Yaskawa INFORM job: DEMO_ROOF_SIDE_0625_3PAINT_9.JBI

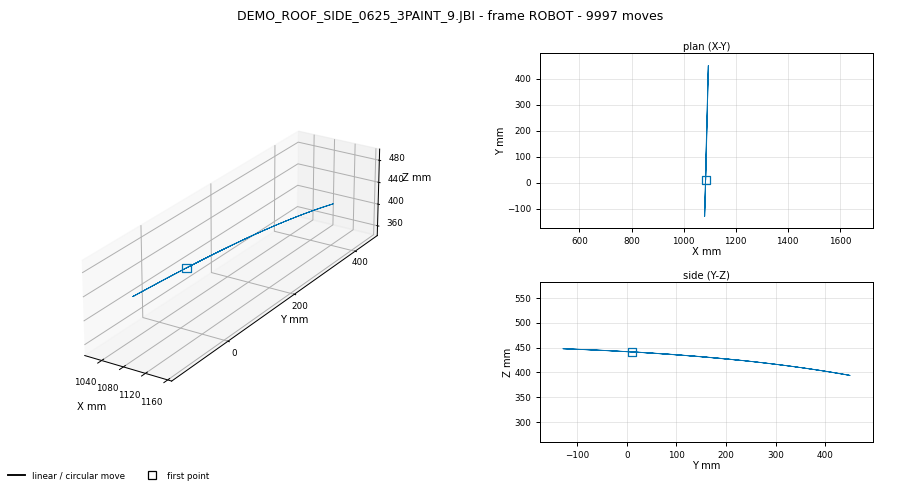
[picture p0: tool path of DEMO_ROOF_SIDE_0625_3PAINT_9.JBI in frame ROBOT, 9997 of 9997 moves have a stored position in this frame; points joined in program order, loops and branches not executed]
/JOB
//NAME DEMO_ROOF_SIDE_0625_3PAINT9
//POS
///NPOS 9997,0,0,0,0,0
///TOOL 0
///USER 0
///POSTYPE ROBOT
///RECTAN
///RCONF 1,0,0,0,0,0,0,0,0,0,0,0,0,0,0,0,0,0,0,0,0,0,0,0
C00000=1085.250,11.093,441.789,174.492,19.107,153.129
C00001=1085.256,11.342,441.774,174.493,19.109,153.129
C00002=1085.262,11.592,441.760,174.496,19.111,153.129
C00003=1085.269,11.841,441.746,174.497,19.113,153.129
C00004=1085.275,12.091,441.732,174.498,19.115,153.129
C00005=1085.280,12.340,441.717,174.500,19.118,153.129
C00006=1085.286,12.590,441.703,174.502,19.119,153.129
C00007=1085.292,12.839,441.688,174.503,19.121,153.129
C00008=1085.298,13.089,441.675,174.505,19.123,153.129
C00009=1085.304,13.338,441.660,174.507,19.125,153.130
C00010=1085.310,13.588,441.646,174.508,19.127,153.130
C00011=1085.315,13.837,441.631,174.509,19.129,153.130
C00012=1085.321,14.087,441.617,174.512,19.131,153.130
C00013=1085.327,14.336,441.602,174.513,19.133,153.130
C00014=1085.333,14.586,441.588,174.514,19.134,153.130
C00015=1085.340,14.863,441.572,174.516,19.137,153.130
C00016=1085.346,15.140,441.555,174.517,19.139,153.130
C00017=1085.352,15.417,441.539,174.520,19.141,153.130
C00018=1085.358,15.693,441.524,174.521,19.143,153.131
C00019=1085.365,15.943,441.509,174.523,19.145,153.131
C00020=1085.370,16.192,441.495,174.524,19.147,153.131
C00021=1085.376,16.443,441.480,174.526,19.149,153.131
C00022=1085.382,16.692,441.465,174.528,19.151,153.131
C00023=1085.387,16.941,441.451,174.529,19.153,153.131
C00024=1085.393,17.191,441.436,174.530,19.155,153.131
C00025=1085.399,17.440,441.422,174.533,19.157,153.131
C00026=1085.405,17.689,441.408,174.534,19.159,153.131
C00027=1085.411,17.939,441.393,174.535,19.161,153.132
C00028=1085.416,18.188,441.378,174.537,19.163,153.132
C00029=1085.422,18.438,441.364,174.539,19.165,153.132
C00030=1085.428,18.687,441.349,174.540,19.167,153.132
C00031=1085.434,18.937,441.334,174.541,19.168,153.132
C00032=1085.440,19.187,441.320,174.544,19.171,153.132
C00033=1085.445,19.436,441.305,174.545,19.173,153.132
C00034=1085.451,19.686,441.290,174.546,19.174,153.132
C00035=1085.457,19.935,441.276,174.548,19.177,153.132
C00036=1085.463,20.185,441.261,174.550,19.178,153.132
C00037=1085.469,20.434,441.247,174.551,19.181,153.133
C00038=1085.474,20.684,441.231,174.553,19.183,153.133
C00039=1085.480,20.933,441.217,174.554,19.185,153.133
C00040=1085.486,21.182,441.203,174.556,19.186,153.133
C00041=1085.491,21.432,441.187,174.558,19.189,153.133
C00042=1085.497,21.681,441.173,174.559,19.191,153.133
C00043=1085.503,21.931,441.158,174.561,19.192,153.133
C00044=1085.509,22.180,441.144,174.563,19.195,153.133
C00045=1085.515,22.430,441.128,174.564,19.196,153.133
C00046=1085.520,22.679,441.114,174.565,19.198,153.134
C00047=1085.527,22.930,441.099,174.568,19.200,153.134
C00048=1085.532,23.179,441.084,174.569,19.202,153.134
C00049=1085.538,23.429,441.069,174.570,19.204,153.134
C00050=1085.544,23.677,441.055,174.572,19.206,153.134
C00051=1085.549,23.927,441.040,174.574,19.208,153.134
C00052=1085.555,24.176,441.025,174.575,19.210,153.134
C00053=1085.561,24.426,441.011,174.577,19.212,153.134
C00054=1085.566,24.676,440.995,174.578,19.214,153.134
C00055=1085.572,24.925,440.981,174.580,19.216,153.135
C00056=1085.578,25.175,440.966,174.582,19.218,153.135
C00057=1085.584,25.424,440.951,174.583,19.220,153.135
C00058=1085.590,25.674,440.936,174.585,19.222,153.135
C00059=1085.596,25.922,440.921,174.587,19.224,153.135
C00060=1085.601,26.172,440.905,174.588,19.226,153.135
C00061=1085.607,26.421,440.891,174.589,19.228,153.135
C00062=1085.613,26.672,440.877,174.592,19.230,153.135
C00063=1085.619,26.922,440.861,174.593,19.232,153.135
C00064=1085.625,27.171,440.847,174.594,19.233,153.135
C00065=1085.630,27.421,440.831,174.596,19.236,153.136
C00066=1085.636,27.670,440.816,174.598,19.237,153.136
C00067=1085.642,27.919,440.801,174.599,19.239,153.136
C00068=1085.647,28.168,440.786,174.601,19.241,153.136
C00069=1085.654,28.418,440.771,174.602,19.243,153.136
C00070=1085.659,28.667,440.756,174.604,19.245,153.136
C00071=1085.665,28.917,440.741,174.606,19.247,153.136
C00072=1085.670,29.166,440.726,174.607,19.249,153.136
C00073=1085.677,29.416,440.711,174.609,19.251,153.136
C00074=1085.682,29.665,440.696,174.611,19.253,153.137
C00075=1085.688,29.915,440.681,174.612,19.255,153.137
C00076=1085.693,30.164,440.666,174.613,19.257,153.137
C00077=1085.700,30.414,440.651,174.616,19.259,153.137
C00078=1085.705,30.664,440.635,174.617,19.261,153.137
C00079=1085.712,30.942,440.618,174.619,19.263,153.137
C00080=1085.718,31.220,440.602,174.620,19.265,153.137
C00081=1085.725,31.498,440.585,174.622,19.268,153.137
C00082=1085.731,31.776,440.568,174.624,19.270,153.137
C00083=1085.736,32.025,440.553,174.626,19.272,153.137
C00084=1085.743,32.275,440.538,174.627,19.274,153.138
C00085=1085.748,32.525,440.522,174.629,19.276,153.138
C00086=1085.754,32.774,440.507,174.631,19.278,153.138
C00087=1085.760,33.023,440.492,174.632,19.279,153.138
C00088=1085.765,33.273,440.476,174.634,19.282,153.138
C00089=1085.771,33.522,440.462,174.636,19.283,153.138
C00090=1085.776,33.772,440.446,174.637,19.285,153.138
C00091=1085.783,34.021,440.431,174.639,19.287,153.138
C00092=1085.788,34.271,440.416,174.640,19.289,153.138
C00093=1085.794,34.520,440.400,174.643,19.291,153.138
C00094=1085.800,34.770,440.385,174.644,19.293,153.139
C00095=1085.806,35.020,440.370,174.645,19.295,153.139
C00096=1085.812,35.268,440.355,174.647,19.298,153.139
C00097=1085.817,35.518,440.339,174.649,19.299,153.139
C00098=1085.822,35.768,440.324,174.650,19.301,153.139
C00099=1085.829,36.017,440.309,174.652,19.303,153.139
C00100=1085.835,36.267,440.293,174.654,19.305,153.139
C00101=1085.840,36.516,440.278,174.655,19.307,153.139
C00102=1085.846,36.766,440.263,174.657,19.309,153.139
C00103=1085.852,37.015,440.247,174.659,19.311,153.139
C00104=1085.858,37.264,440.232,174.661,19.313,153.139
C00105=1085.863,37.514,440.217,174.662,19.315,153.140
C00106=1085.870,37.764,440.202,174.663,19.316,153.140
C00107=1085.875,38.012,440.186,174.666,19.319,153.140
C00108=1085.881,38.262,440.170,174.667,19.320,153.140
C00109=1085.886,38.512,440.155,174.668,19.322,153.140
C00110=1085.893,38.760,440.139,174.671,19.324,153.140
C00111=1085.898,39.010,440.124,174.672,19.326,153.140
C00112=1085.904,39.260,440.108,174.674,19.328,153.140
C00113=1085.909,39.509,440.092,174.675,19.330,153.140
C00114=1085.915,39.759,440.077,174.677,19.332,153.140
C00115=1085.921,40.009,440.062,174.679,19.334,153.141
C00116=1085.927,40.257,440.046,174.680,19.336,153.141
C00117=1085.932,40.507,440.030,174.682,19.338,153.141
C00118=1085.938,40.757,440.015,174.684,19.340,153.141
C00119=1085.944,41.006,440.000,174.685,19.342,153.141
C00120=1085.950,41.256,439.984,174.687,19.344,153.141
C00121=1085.955,41.506,439.968,174.688,19.346,153.141
C00122=1085.961,41.754,439.953,174.690,19.348,153.141
C00123=1085.966,42.004,439.937,174.692,19.350,153.141
C00124=1085.972,42.253,439.921,174.693,19.352,153.141
C00125=1085.978,42.502,439.906,174.695,19.354,153.142
C00126=1085.984,42.752,439.890,174.697,19.356,153.142
C00127=1085.990,43.002,439.874,174.698,19.357,153.142
C00128=1085.995,43.252,439.859,174.700,19.360,153.142
C00129=1086.001,43.500,439.843,174.702,19.361,153.142
C00130=1086.007,43.750,439.828,174.704,19.364,153.142
C00131=1086.013,43.999,439.812,174.705,19.365,153.142
C00132=1086.018,44.249,439.797,174.707,19.367,153.142
C00133=1086.024,44.498,439.780,174.709,19.369,153.142
C00134=1086.030,44.748,439.765,174.710,19.371,153.142
C00135=1086.035,44.997,439.749,174.712,19.373,153.142
C00136=1086.041,45.247,439.733,174.714,19.375,153.143
C00137=1086.047,45.496,439.717,174.715,19.377,153.143
C00138=1086.052,45.746,439.702,174.717,19.379,153.143
C00139=1086.058,45.995,439.686,174.719,19.381,153.143
C00140=1086.063,46.245,439.670,174.721,19.383,153.143
C00141=1086.069,46.494,439.654,174.722,19.385,153.143
C00142=1086.074,46.743,439.639,174.723,19.387,153.143
C00143=1086.081,47.022,439.621,174.726,19.389,153.143
C00144=1086.087,47.300,439.603,174.728,19.391,153.143
C00145=1086.092,47.578,439.585,174.729,19.393,153.144
C00146=1086.100,47.857,439.568,174.731,19.396,153.144
C00147=1086.105,48.105,439.552,174.733,19.398,153.144
C00148=1086.111,48.355,439.535,174.735,19.400,153.144
C00149=1086.117,48.605,439.520,174.736,19.402,153.144
C00150=1086.123,48.854,439.504,174.738,19.404,153.144
C00151=1086.127,49.103,439.487,174.740,19.406,153.144
C00152=1086.133,49.353,439.472,174.742,19.408,153.144
C00153=1086.139,49.602,439.455,174.743,19.410,153.144
C00154=1086.144,49.852,439.440,174.745,19.411,153.144
C00155=1086.150,50.102,439.424,174.747,19.413,153.144
C00156=1086.156,50.350,439.408,174.748,19.415,153.145
C00157=1086.161,50.600,439.392,174.750,19.417,153.145
C00158=1086.167,50.850,439.376,174.752,19.419,153.145
C00159=1086.173,51.099,439.360,174.753,19.421,153.145
C00160=1086.179,51.348,439.343,174.755,19.423,153.145
C00161=1086.184,51.598,439.328,174.757,19.425,153.145
C00162=1086.190,51.847,439.312,174.759,19.427,153.145
C00163=1086.196,52.096,439.296,174.760,19.429,153.145
C00164=1086.202,52.346,439.279,174.762,19.431,153.145
C00165=1086.207,52.596,439.263,174.764,19.433,153.145
C00166=1086.212,52.845,439.247,174.765,19.434,153.145
C00167=1086.218,53.094,439.231,174.767,19.436,153.145
C00168=1086.224,53.343,439.215,174.769,19.438,153.146
C00169=1086.230,53.593,439.199,174.771,19.440,153.146
C00170=1086.236,53.843,439.183,174.772,19.442,153.146
C00171=1086.242,54.092,439.167,174.774,19.444,153.146
C00172=1086.248,54.341,439.151,174.776,19.446,153.146
C00173=1086.253,54.590,439.135,174.777,19.447,153.146
C00174=1086.258,54.840,439.119,174.779,19.450,153.146
C00175=1086.264,55.089,439.102,174.781,19.451,153.146
C00176=1086.270,55.339,439.086,174.783,19.454,153.146
C00177=1086.276,55.588,439.070,174.784,19.455,153.146
C00178=1086.282,55.838,439.054,174.787,19.457,153.146
C00179=1086.288,56.087,439.037,174.788,19.460,153.146
C00180=1086.293,56.337,439.022,174.789,19.461,153.146
C00181=1086.299,56.587,439.005,174.792,19.463,153.146
C00182=1086.305,56.836,438.989,174.793,19.465,153.146
C00183=1086.310,57.085,438.973,174.795,19.467,153.147
C00184=1086.316,57.334,438.956,174.797,19.469,153.147
C00185=1086.322,57.583,438.940,174.799,19.471,153.147
C00186=1086.328,57.833,438.924,174.800,19.473,153.147
C00187=1086.333,58.082,438.907,174.802,19.474,153.147
C00188=1086.339,58.332,438.891,174.804,19.476,153.147
C00189=1086.345,58.581,438.875,174.805,19.478,153.147
C00190=1086.351,58.830,438.858,174.808,19.480,153.147
C00191=1086.357,59.080,438.842,174.809,19.482,153.147
C00192=1086.362,59.329,438.825,174.811,19.484,153.147
C00193=1086.368,59.579,438.809,174.813,19.486,153.147
C00194=1086.374,59.828,438.793,174.814,19.487,153.147
C00195=1086.380,60.077,438.776,174.816,19.489,153.147
C00196=1086.386,60.327,438.760,174.818,19.491,153.147
C00197=1086.391,60.576,438.743,174.820,19.493,153.148
C00198=1086.397,60.826,438.727,174.821,19.495,153.148
C00199=1086.403,61.075,438.711,174.824,19.497,153.148
C00200=1086.409,61.324,438.695,174.825,19.498,153.148
C00201=1086.415,61.574,438.678,174.827,19.501,153.148
C00202=1086.420,61.823,438.661,174.829,19.502,153.148
C00203=1086.426,62.073,438.645,174.830,19.504,153.148
C00204=1086.432,62.322,438.629,174.832,19.506,153.148
C00205=1086.438,62.571,438.613,174.834,19.507,153.148
C00206=1086.443,62.821,438.596,174.836,19.510,153.148
C00207=1086.451,63.099,438.578,174.838,19.512,153.148
C00208=1086.457,63.376,438.559,174.840,19.513,153.148
C00209=1086.463,63.655,438.541,174.842,19.516,153.148
C00210=1086.470,63.933,438.523,174.844,19.518,153.148
C00211=1086.476,64.182,438.506,174.845,19.519,153.148
C00212=1086.481,64.432,438.489,174.848,19.521,153.148
C00213=1086.487,64.681,438.473,174.849,19.523,153.149
C00214=1086.492,64.930,438.456,174.851,19.525,153.149
C00215=1086.498,65.180,438.439,174.853,19.527,153.149
C00216=1086.504,65.429,438.423,174.855,19.529,153.149
C00217=1086.509,65.679,438.406,174.856,19.531,153.149
C00218=1086.515,65.928,438.390,174.858,19.532,153.149
C00219=1086.521,66.177,438.372,174.860,19.534,153.149
C00220=1086.527,66.426,438.356,174.862,19.536,153.149
C00221=1086.532,66.676,438.339,174.864,19.538,153.149
C00222=1086.538,66.925,438.323,174.865,19.540,153.149
C00223=1086.544,67.175,438.307,174.867,19.542,153.149
C00224=1086.550,67.424,438.289,174.869,19.543,153.149
C00225=1086.556,67.674,438.273,174.871,19.545,153.149
C00226=1086.561,67.923,438.256,174.872,19.547,153.149
C00227=1086.567,68.173,438.240,174.875,19.549,153.149
C00228=1086.573,68.422,438.222,174.876,19.551,153.149
C00229=1086.579,68.671,438.206,174.878,19.553,153.149
C00230=1086.584,68.921,438.189,174.880,19.554,153.149
C00231=1086.590,69.170,438.172,174.882,19.557,153.150
C00232=1086.595,69.419,438.155,174.883,19.558,153.150
C00233=1086.601,69.669,438.139,174.885,19.560,153.150
C00234=1086.607,69.918,438.121,174.887,19.562,153.150
C00235=1086.612,70.167,438.104,174.889,19.564,153.150
C00236=1086.618,70.417,438.088,174.891,19.566,153.150
C00237=1086.624,70.666,438.071,174.892,19.568,153.150
C00238=1086.629,70.915,438.054,174.895,19.570,153.150
C00239=1086.635,71.165,438.037,174.896,19.571,153.150
C00240=1086.641,71.414,438.020,174.898,19.573,153.150
C00241=1086.647,71.664,438.003,174.900,19.575,153.150
C00242=1086.652,71.913,437.986,174.902,19.577,153.150
C00243=1086.658,72.162,437.969,174.903,19.579,153.150
C00244=1086.663,72.412,437.953,174.906,19.581,153.150
C00245=1086.669,72.661,437.935,174.907,19.582,153.150
C00246=1086.675,72.910,437.919,174.909,19.585,153.150
C00247=1086.680,73.159,437.901,174.911,19.586,153.150
C00248=1086.686,73.409,437.884,174.913,19.588,153.150
C00249=1086.692,73.658,437.867,174.914,19.590,153.151
C00250=1086.698,73.908,437.850,174.917,19.592,153.151
C00251=1086.703,74.158,437.833,174.918,19.593,153.151
C00252=1086.709,74.406,437.816,174.921,19.595,153.151
C00253=1086.714,74.656,437.799,174.922,19.597,153.151
C00254=1086.720,74.905,437.782,174.924,19.599,153.151
C00255=1086.726,75.154,437.766,174.926,19.601,153.151
C00256=1086.732,75.404,437.748,174.928,19.603,153.151
C00257=1086.737,75.654,437.731,174.929,19.604,153.151
C00258=1086.743,75.902,437.714,174.932,19.606,153.151
C00259=1086.749,76.152,437.696,174.933,19.608,153.151
C00260=1086.754,76.401,437.679,174.935,19.610,153.151
C00261=1086.760,76.650,437.663,174.937,19.612,153.151
C00262=1086.766,76.900,437.645,174.939,19.614,153.151
C00263=1086.772,77.149,437.628,174.940,19.615,153.151
C00264=1086.777,77.399,437.611,174.943,19.617,153.151
C00265=1086.783,77.648,437.594,174.944,19.619,153.151
C00266=1086.789,77.897,437.576,174.947,19.621,153.151
C00267=1086.795,78.147,437.559,174.948,19.622,153.151
C00268=1086.800,78.396,437.542,174.950,19.624,153.151
C00269=1086.806,78.646,437.525,174.952,19.626,153.151
C00270=1086.812,78.895,437.508,174.954,19.628,153.151
C00271=1086.818,79.173,437.488,174.956,19.630,153.151
C00272=1086.824,79.450,437.469,174.958,19.632,153.152
C00273=1086.830,79.728,437.450,174.960,19.634,153.152
C00274=1086.836,80.007,437.430,174.962,19.636,153.152
C00275=1086.843,80.256,437.413,174.964,19.637,153.152
C00276=1086.848,80.505,437.396,174.966,19.640,153.152
C00277=1086.853,80.754,437.379,174.967,19.641,153.152
C00278=1086.859,81.003,437.361,174.970,19.643,153.152
C00279=1086.865,81.253,437.343,174.972,19.645,153.152
C00280=1086.870,81.503,437.327,174.973,19.647,153.152
C00281=1086.876,81.752,437.309,174.976,19.649,153.152
C00282=1086.881,82.001,437.291,174.977,19.650,153.152
C00283=1086.887,82.251,437.273,174.979,19.652,153.152
C00284=1086.893,82.500,437.257,174.981,19.654,153.152
C00285=1086.898,82.749,437.239,174.983,19.656,153.152
C00286=1086.904,82.998,437.222,174.985,19.657,153.152
C00287=1086.910,83.247,437.205,174.987,19.659,153.152
C00288=1086.916,83.497,437.187,174.988,19.661,153.152
C00289=1086.921,83.747,437.170,174.991,19.663,153.152
C00290=1086.927,83.996,437.152,174.992,19.665,153.152
C00291=1086.933,84.245,437.134,174.994,19.667,153.152
C00292=1086.938,84.494,437.117,174.996,19.668,153.152
C00293=1086.944,84.743,437.099,174.998,19.670,153.152
C00294=1086.949,84.992,437.082,175.000,19.672,153.152
C00295=1086.955,85.243,437.064,175.002,19.674,153.152
C00296=1086.961,85.492,437.047,175.003,19.675,153.152
C00297=1086.966,85.741,437.029,175.006,19.677,153.152
C00298=1086.972,85.990,437.012,175.007,19.679,153.152
C00299=1086.978,86.240,436.994,175.009,19.681,153.152
C00300=1086.983,86.489,436.976,175.012,19.683,153.152
C00301=1086.989,86.738,436.959,175.013,19.684,153.153
C00302=1086.995,86.987,436.941,175.016,19.686,153.152
C00303=1087.000,87.237,436.924,175.017,19.687,153.152
C00304=1087.006,87.486,436.906,175.020,19.689,153.152
C00305=1087.012,87.736,436.888,175.021,19.691,153.153
C00306=1087.017,87.985,436.871,175.023,19.693,153.153
C00307=1087.023,88.234,436.853,175.025,19.694,153.153
C00308=1087.029,88.484,436.835,175.027,19.696,153.153
C00309=1087.035,88.733,436.818,175.029,19.698,153.153
C00310=1087.040,88.982,436.800,175.031,19.700,153.153
C00311=1087.046,89.232,436.782,175.032,19.701,153.153
C00312=1087.052,89.481,436.765,175.035,19.703,153.153
C00313=1087.058,89.730,436.747,175.037,19.705,153.153
C00314=1087.063,89.979,436.729,175.039,19.707,153.153
C00315=1087.069,90.228,436.712,175.041,19.708,153.153
C00316=1087.075,90.478,436.694,175.043,19.710,153.153
C00317=1087.080,90.727,436.676,175.045,19.712,153.153
C00318=1087.087,90.977,436.658,175.046,19.713,153.153
C00319=1087.092,91.226,436.641,175.049,19.715,153.153
C00320=1087.097,91.475,436.622,175.050,19.717,153.153
C00321=1087.103,91.724,436.604,175.052,19.719,153.153
C00322=1087.109,91.973,436.586,175.055,19.721,153.153
C00323=1087.114,92.223,436.569,175.056,19.722,153.153
C00324=1087.120,92.472,436.551,175.059,19.724,153.153
C00325=1087.125,92.722,436.532,175.060,19.726,153.153
C00326=1087.131,92.971,436.515,175.062,19.728,153.153
C00327=1087.137,93.220,436.497,175.064,19.729,153.153
C00328=1087.142,93.469,436.479,175.066,19.731,153.153
C00329=1087.148,93.718,436.461,175.068,19.732,153.153
C00330=1087.154,93.968,436.443,175.070,19.734,153.153
C00331=1087.159,94.217,436.425,175.072,19.736,153.153
C00332=1087.165,94.467,436.407,175.074,19.738,153.153
C00333=1087.170,94.716,436.389,175.076,19.740,153.153
C00334=1087.176,94.965,436.371,175.078,19.741,153.153
C00335=1087.182,95.243,436.351,175.080,19.743,153.153
C00336=1087.188,95.521,436.331,175.082,19.745,153.153
C00337=1087.195,95.799,436.311,175.085,19.747,153.153
C00338=1087.202,96.077,436.290,175.087,19.749,153.153
C00339=1087.206,96.327,436.272,175.088,19.751,153.153
C00340=1087.212,96.576,436.255,175.091,19.752,153.153
C00341=1087.218,96.825,436.236,175.092,19.754,153.153
C00342=1087.224,97.074,436.219,175.095,19.756,153.153
C00343=1087.229,97.324,436.200,175.097,19.758,153.153
C00344=1087.235,97.572,436.182,175.099,19.759,153.153
C00345=1087.241,97.822,436.164,175.101,19.761,153.153
C00346=1087.246,98.071,436.146,175.103,19.762,153.153
C00347=1087.252,98.321,436.127,175.105,19.764,153.153
C00348=1087.258,98.570,436.109,175.107,19.766,153.153
C00349=1087.263,98.820,436.091,175.109,19.768,153.153
C00350=1087.269,99.068,436.073,175.111,19.769,153.153
C00351=1087.275,99.318,436.055,175.113,19.771,153.153
C00352=1087.281,99.567,436.037,175.115,19.773,153.153
C00353=1087.287,99.816,436.018,175.117,19.774,153.153
C00354=1087.292,100.065,436.000,175.119,19.776,153.153
C00355=1087.298,100.315,435.982,175.121,19.778,153.153
C00356=1087.303,100.564,435.963,175.123,19.779,153.153
C00357=1087.309,100.814,435.946,175.125,19.781,153.153
C00358=1087.314,101.062,435.927,175.127,19.782,153.153
C00359=1087.321,101.312,435.909,175.129,19.784,153.153
C00360=1087.326,101.561,435.891,175.132,19.786,153.153
C00361=1087.332,101.811,435.872,175.133,19.788,153.153
C00362=1087.337,102.060,435.854,175.135,19.790,153.153
C00363=1087.343,102.309,435.835,175.137,19.791,153.153
C00364=1087.349,102.558,435.818,175.139,19.793,153.153
C00365=1087.354,102.807,435.798,175.142,19.795,153.153
C00366=1087.360,103.057,435.781,175.143,19.796,153.153
C00367=1087.365,103.306,435.761,175.145,19.798,153.153
C00368=1087.371,103.555,435.744,175.147,19.799,153.153
C00369=1087.377,103.804,435.725,175.150,19.801,153.153
C00370=1087.381,104.054,435.707,175.152,19.803,153.153
C00371=1087.388,104.303,435.688,175.153,19.804,153.153
C00372=1087.393,104.552,435.670,175.156,19.806,153.153
C00373=1087.399,104.801,435.651,175.157,19.807,153.153
C00374=1087.404,105.051,435.633,175.160,19.809,153.153
C00375=1087.410,105.300,435.614,175.162,19.811,153.153
C00376=1087.416,105.549,435.595,175.164,19.812,153.153
C00377=1087.421,105.798,435.577,175.166,19.814,153.153
C00378=1087.427,106.048,435.558,175.167,19.816,153.153
C00379=1087.432,106.297,435.540,175.170,19.817,153.153
C00380=1087.438,106.546,435.521,175.172,19.819,153.153
C00381=1087.444,106.796,435.502,175.174,19.821,153.153
C00382=1087.450,107.045,435.485,175.176,19.822,153.153
C00383=1087.455,107.294,435.465,175.178,19.824,153.153
C00384=1087.461,107.543,435.448,175.180,19.826,153.153
C00385=1087.466,107.793,435.429,175.183,19.827,153.153
C00386=1087.472,108.042,435.409,175.184,19.829,153.153
C00387=1087.478,108.291,435.392,175.187,19.831,153.153
C00388=1087.483,108.540,435.372,175.189,19.832,153.152
C00389=1087.489,108.789,435.354,175.191,19.834,153.153
C00390=1087.495,109.038,435.335,175.193,19.836,153.153
C00391=1087.500,109.288,435.316,175.195,19.837,153.152
C00392=1087.506,109.537,435.298,175.197,19.839,153.152
C00393=1087.512,109.786,435.279,175.199,19.840,153.152
C00394=1087.518,110.036,435.261,175.201,19.842,153.152
C00395=1087.523,110.285,435.242,175.203,19.844,153.152
C00396=1087.529,110.534,435.223,175.206,19.845,153.152
C00397=1087.535,110.783,435.204,175.207,19.847,153.152
C00398=1087.540,111.033,435.186,175.210,19.848,153.152
C00399=1087.546,111.311,435.164,175.212,19.850,153.152
C00400=1087.553,111.589,435.144,175.215,19.852,153.152
C00401=1087.559,111.866,435.123,175.217,19.854,153.152
C00402=1087.566,112.145,435.102,175.219,19.856,153.152
C00403=1087.571,112.394,435.083,175.221,19.857,153.152
C00404=1087.577,112.643,435.064,175.223,19.859,153.152
C00405=1087.582,112.893,435.045,175.225,19.860,153.152
C00406=1087.588,113.141,435.026,175.227,19.862,153.152
C00407=1087.594,113.390,435.007,175.230,19.864,153.152
C00408=1087.599,113.640,434.989,175.231,19.865,153.152
C00409=1087.605,113.890,434.969,175.234,19.867,153.152
C00410=1087.611,114.138,434.951,175.236,19.869,153.152
C00411=1087.616,114.388,434.932,175.238,19.870,153.152
C00412=1087.622,114.637,434.913,175.240,19.872,153.152
C00413=1087.627,114.886,434.894,175.243,19.873,153.152
C00414=1087.633,115.135,434.875,175.244,19.875,153.152
C00415=1087.638,115.385,434.855,175.247,19.877,153.152
C00416=1087.644,115.634,434.836,175.249,19.878,153.152
C00417=1087.649,115.883,434.817,175.251,19.880,153.152
C00418=1087.655,116.132,434.798,175.253,19.882,153.152
C00419=1087.660,116.381,434.779,175.255,19.883,153.152
C00420=1087.666,116.631,434.760,175.257,19.885,153.152
C00421=1087.671,116.880,434.741,175.259,19.886,153.151
C00422=1087.676,117.129,434.722,175.262,19.888,153.151
C00423=1087.682,117.378,434.702,175.263,19.890,153.152
C00424=1087.689,117.627,434.684,175.266,19.891,153.151
C00425=1087.694,117.876,434.665,175.268,19.893,153.151
C00426=1087.699,118.125,434.646,175.270,19.894,153.151
C00427=1087.705,118.375,434.626,175.272,19.896,153.151
C00428=1087.711,118.624,434.607,175.275,19.897,153.151
C00429=1087.716,118.873,434.588,175.276,19.899,153.151
C00430=1087.721,119.122,434.569,175.279,19.900,153.151
C00431=1087.727,119.372,434.550,175.281,19.902,153.151
C00432=1087.733,119.621,434.531,175.283,19.903,153.151
C00433=1087.738,119.870,434.512,175.285,19.905,153.151
C00434=1087.744,120.120,434.492,175.288,19.907,153.151
C00435=1087.749,120.369,434.473,175.289,19.908,153.151
C00436=1087.755,120.618,434.454,175.292,19.910,153.151
C00437=1087.760,120.866,434.434,175.294,19.912,153.151
C00438=1087.766,121.116,434.415,175.296,19.913,153.151
C00439=1087.772,121.365,434.396,175.298,19.915,153.151
C00440=1087.777,121.615,434.377,175.301,19.916,153.151
C00441=1087.782,121.864,434.357,175.302,19.918,153.151
C00442=1087.788,122.113,434.338,175.305,19.919,153.151
C00443=1087.793,122.362,434.318,175.307,19.921,153.151
C00444=1087.799,122.612,434.299,175.309,19.922,153.151
C00445=1087.805,122.861,434.280,175.311,19.924,153.151
C00446=1087.811,123.110,434.260,175.314,19.926,153.150
C00447=1087.816,123.358,434.241,175.315,19.927,153.150
C00448=1087.822,123.608,434.221,175.318,19.929,153.150
C00449=1087.827,123.857,434.202,175.320,19.930,153.150
C00450=1087.833,124.107,434.183,175.322,19.932,153.150
C00451=1087.839,124.356,434.163,175.324,19.933,153.150
C00452=1087.845,124.605,434.144,175.327,19.935,153.150
C00453=1087.850,124.854,434.125,175.329,19.937,153.150
C00454=1087.855,125.103,434.106,175.331,19.938,153.150
C00455=1087.861,125.352,434.086,175.333,19.940,153.150
C00456=1087.867,125.601,434.066,175.336,19.941,153.150
C00457=1087.872,125.851,434.047,175.337,19.942,153.150
C00458=1087.878,126.100,434.027,175.340,19.944,153.150
C00459=1087.884,126.349,434.007,175.342,19.946,153.150
C00460=1087.889,126.599,433.988,175.344,19.947,153.150
C00461=1087.895,126.848,433.968,175.346,19.949,153.150
C00462=1087.901,127.096,433.949,175.349,19.950,153.149
C00463=1087.907,127.375,433.927,175.351,19.952,153.149
C00464=1087.914,127.653,433.906,175.354,19.954,153.149
C00465=1087.920,127.930,433.884,175.356,19.955,153.149
C00466=1087.926,128.208,433.862,175.359,19.957,153.149
C00467=1087.931,128.458,433.842,175.361,19.959,153.149
C00468=1087.937,128.707,433.822,175.363,19.960,153.149
C00469=1087.943,128.956,433.803,175.365,19.961,153.149
C00470=1087.949,129.206,433.783,175.368,19.963,153.149
C00471=1087.955,129.454,433.763,175.369,19.964,153.149
C00472=1087.960,129.704,433.744,175.372,19.965,153.149
C00473=1087.966,129.953,433.724,175.375,19.967,153.149
C00474=1087.971,130.202,433.704,175.377,19.968,153.148
C00475=1087.977,130.451,433.684,175.379,19.970,153.148
C00476=1087.983,130.701,433.665,175.381,19.971,153.148
C00477=1087.989,130.950,433.645,175.384,19.973,153.148
C00478=1087.995,131.199,433.626,175.385,19.974,153.148
C00479=1088.000,131.448,433.605,175.388,19.975,153.148
C00480=1088.006,131.697,433.585,175.390,19.977,153.148
C00481=1088.012,131.946,433.566,175.393,19.979,153.148
C00482=1088.018,132.195,433.546,175.395,19.980,153.148
C00483=1088.023,132.445,433.527,175.397,19.981,153.148
C00484=1088.029,132.694,433.506,175.400,19.983,153.148
C00485=1088.034,132.943,433.487,175.401,19.984,153.148
C00486=1088.040,133.192,433.467,175.404,19.986,153.147
C00487=1088.046,133.441,433.447,175.406,19.987,153.147
C00488=1088.051,133.690,433.427,175.409,19.989,153.147
C00489=1088.057,133.940,433.407,175.410,19.990,153.147
C00490=1088.063,134.188,433.387,175.413,19.992,153.147
C00491=1088.067,134.438,433.367,175.416,19.993,153.147
C00492=1088.073,134.687,433.347,175.418,19.995,153.147
C00493=1088.079,134.936,433.327,175.420,19.996,153.147
C00494=1088.084,135.186,433.307,175.422,19.998,153.147
C00495=1088.090,135.434,433.287,175.425,19.999,153.147
C00496=1088.096,135.683,433.267,175.427,20.001,153.147
C00497=1088.101,135.933,433.248,175.429,20.002,153.147
C00498=1088.107,136.182,433.228,175.431,20.004,153.146
C00499=1088.113,136.431,433.207,175.434,20.005,153.146
C00500=1088.119,136.680,433.187,175.436,20.007,153.146
C00501=1088.124,136.929,433.167,175.438,20.008,153.146
C00502=1088.130,137.178,433.147,175.440,20.010,153.146
C00503=1088.135,137.427,433.127,175.443,20.011,153.146
C00504=1088.141,137.676,433.107,175.446,20.013,153.146
C00505=1088.146,137.926,433.088,175.447,20.014,153.146
C00506=1088.152,138.175,433.067,175.450,20.015,153.146
C00507=1088.158,138.424,433.047,175.452,20.017,153.146
C00508=1088.163,138.673,433.027,175.455,20.019,153.146
C00509=1088.169,138.921,433.007,175.456,20.020,153.146
C00510=1088.174,139.171,432.986,175.459,20.021,153.145
C00511=1088.180,139.420,432.967,175.462,20.022,153.145
C00512=1088.185,139.669,432.946,175.464,20.024,153.145
C00513=1088.190,139.918,432.926,175.466,20.025,153.145
C00514=1088.197,140.168,432.905,175.468,20.026,153.145
C00515=1088.202,140.417,432.885,175.471,20.028,153.145
C00516=1088.208,140.666,432.865,175.473,20.030,153.145
C00517=1088.214,140.915,432.844,175.475,20.031,153.145
C00518=1088.220,141.164,432.824,175.478,20.032,153.145
C00519=1088.225,141.413,432.804,175.480,20.034,153.144
C00520=1088.230,141.663,432.784,175.483,20.035,153.144
C00521=1088.236,141.911,432.764,175.485,20.037,153.144
C00522=1088.241,142.160,432.743,175.487,20.038,153.144
C00523=1088.246,142.410,432.723,175.489,20.040,153.144
C00524=1088.253,142.659,432.703,175.492,20.041,153.144
C00525=1088.258,142.908,432.682,175.494,20.043,153.144
C00526=1088.263,143.157,432.661,175.496,20.044,153.144
C00527=1088.270,143.435,432.639,175.499,20.046,153.144
C00528=1088.276,143.713,432.616,175.502,20.047,153.144
C00529=1088.282,143.990,432.593,175.505,20.049,153.143
C00530=1088.289,144.268,432.570,175.507,20.050,153.143
C00531=1088.295,144.518,432.550,175.510,20.052,153.143
C00532=1088.300,144.767,432.529,175.511,20.053,153.143
C00533=1088.306,145.016,432.509,175.514,20.055,153.143
C00534=1088.311,145.265,432.489,175.516,20.056,153.143
C00535=1088.316,145.514,432.468,175.519,20.058,153.143
C00536=1088.322,145.763,432.448,175.521,20.059,153.143
C00537=1088.328,146.013,432.427,175.523,20.060,153.143
C00538=1088.333,146.262,432.407,175.526,20.062,153.143
C00539=1088.339,146.511,432.386,175.528,20.063,153.142
C00540=1088.345,146.759,432.365,175.531,20.065,153.142
C00541=1088.350,147.008,432.345,175.533,20.066,153.142
C00542=1088.356,147.258,432.324,175.535,20.067,153.142
C00543=1088.362,147.507,432.304,175.538,20.069,153.142
C00544=1088.367,147.756,432.283,175.540,20.070,153.142
C00545=1088.373,148.005,432.263,175.543,20.072,153.142
C00546=1088.378,148.254,432.241,175.545,20.073,153.142
C00547=1088.385,148.503,432.221,175.547,20.074,153.141
C00548=1088.390,148.752,432.201,175.550,20.075,153.141
C00549=1088.395,149.001,432.180,175.552,20.077,153.141
C00550=1088.401,149.250,432.159,175.555,20.078,153.141
C00551=1088.406,149.499,432.138,175.557,20.080,153.141
C00552=1088.412,149.749,432.117,175.560,20.081,153.141
C00553=1088.417,149.998,432.097,175.562,20.082,153.141
C00554=1088.424,150.246,432.076,175.564,20.084,153.141
C00555=1088.429,150.495,432.056,175.567,20.085,153.141
C00556=1088.435,150.745,432.035,175.569,20.087,153.140
C00557=1088.440,150.994,432.014,175.572,20.088,153.140
C00558=1088.445,151.243,431.993,175.574,20.089,153.140
C00559=1088.451,151.492,431.972,175.576,20.091,153.140
C00560=1088.457,151.742,431.951,175.579,20.092,153.140
C00561=1088.462,151.990,431.930,175.581,20.094,153.140
C00562=1088.467,152.239,431.909,175.584,20.095,153.140
C00563=1088.473,152.488,431.889,175.587,20.096,153.139
C00564=1088.480,152.737,431.868,175.588,20.097,153.139
C00565=1088.485,152.986,431.847,175.591,20.099,153.139
C00566=1088.490,153.235,431.826,175.593,20.100,153.139
C00567=1088.496,153.485,431.805,175.596,20.102,153.139
C00568=1088.501,153.734,431.785,175.599,20.103,153.139
C00569=1088.507,153.982,431.763,175.601,20.105,153.139
C00570=1088.512,154.231,431.743,175.603,20.106,153.139
C00571=1088.518,154.481,431.721,175.605,20.107,153.139
C00572=1088.524,154.730,431.701,175.608,20.109,153.138
C00573=1088.529,154.978,431.679,175.610,20.110,153.138
C00574=1088.535,155.228,431.658,175.613,20.112,153.138
C00575=1088.541,155.477,431.637,175.616,20.113,153.138
C00576=1088.546,155.726,431.617,175.618,20.114,153.138
C00577=1088.552,155.975,431.595,175.620,20.115,153.138
C00578=1088.557,156.224,431.574,175.623,20.117,153.138
C00579=1088.563,156.473,431.553,175.625,20.118,153.138
C00580=1088.569,156.722,431.532,175.628,20.120,153.137
C00581=1088.574,156.971,431.511,175.630,20.121,153.137
C00582=1088.579,157.220,431.490,175.633,20.123,153.137
C00583=1088.585,157.470,431.468,175.635,20.124,153.137
C00584=1088.590,157.719,431.448,175.637,20.125,153.137
C00585=1088.596,157.967,431.426,175.640,20.126,153.137
C00586=1088.602,158.216,431.405,175.643,20.128,153.137
C00587=1088.607,158.466,431.384,175.645,20.129,153.136
C00588=1088.613,158.715,431.362,175.648,20.130,153.136
C00589=1088.619,158.963,431.341,175.650,20.132,153.136
C00590=1088.624,159.212,431.321,175.653,20.133,153.136
C00591=1088.631,159.490,431.297,175.656,20.134,153.136
C00592=1088.636,159.768,431.273,175.658,20.136,153.136
C00593=1088.643,160.046,431.249,175.661,20.137,153.136
C00594=1088.649,160.323,431.225,175.663,20.139,153.135
C00595=1088.655,160.573,431.205,175.666,20.140,153.135
C00596=1088.660,160.821,431.183,175.669,20.141,153.135
C00597=1088.666,161.070,431.162,175.671,20.143,153.135
C00598=1088.671,161.319,431.140,175.674,20.144,153.135
C00599=1088.677,161.569,431.119,175.676,20.146,153.135
C00600=1088.683,161.817,431.098,175.679,20.147,153.134
C00601=1088.688,162.066,431.076,175.681,20.148,153.134
C00602=1088.694,162.315,431.054,175.683,20.149,153.134
C00603=1088.699,162.565,431.033,175.686,20.151,153.134
C00604=1088.704,162.814,431.011,175.688,20.152,153.134
C00605=1088.710,163.063,430.990,175.691,20.154,153.134
C00606=1088.716,163.311,430.969,175.694,20.155,153.134
C00607=1088.721,163.561,430.946,175.696,20.157,153.134
C00608=1088.726,163.810,430.926,175.699,20.158,153.134
C00609=1088.731,164.058,430.904,175.701,20.160,153.133
C00610=1088.737,164.308,430.882,175.704,20.161,153.133
C00611=1088.742,164.557,430.861,175.706,20.162,153.133
C00612=1088.748,164.806,430.839,175.708,20.163,153.133
C00613=1088.754,165.054,430.818,175.711,20.165,153.133
C00614=1088.759,165.303,430.796,175.713,20.166,153.133
C00615=1088.764,165.553,430.775,175.716,20.168,153.133
C00616=1088.769,165.802,430.753,175.719,20.169,153.132
C00617=1088.775,166.051,430.731,175.721,20.170,153.132
C00618=1088.780,166.300,430.710,175.724,20.172,153.132
C00619=1088.786,166.549,430.688,175.727,20.173,153.132
C00620=1088.791,166.798,430.666,175.729,20.175,153.132
C00621=1088.797,167.047,430.644,175.732,20.176,153.132
C00622=1088.803,167.295,430.623,175.734,20.177,153.132
C00623=1088.808,167.544,430.601,175.736,20.178,153.131
C00624=1088.814,167.793,430.580,175.739,20.180,153.131
C00625=1088.819,168.042,430.558,175.741,20.181,153.131
C00626=1088.825,168.291,430.536,175.744,20.182,153.131
C00627=1088.830,168.540,430.514,175.747,20.183,153.131
C00628=1088.836,168.789,430.493,175.749,20.185,153.131
C00629=1088.841,169.038,430.471,175.752,20.186,153.131
C00630=1088.847,169.288,430.449,175.754,20.188,153.130
C00631=1088.852,169.536,430.427,175.757,20.189,153.130
C00632=1088.858,169.786,430.406,175.760,20.190,153.130
C00633=1088.863,170.035,430.383,175.762,20.192,153.130
C00634=1088.869,170.284,430.362,175.765,20.193,153.130
C00635=1088.875,170.532,430.339,175.768,20.194,153.130
C00636=1088.879,170.781,430.317,175.769,20.195,153.129
C00637=1088.886,171.030,430.296,175.772,20.197,153.129
C00638=1088.890,171.279,430.274,175.775,20.198,153.129
C00639=1088.897,171.528,430.252,175.777,20.199,153.129
C00640=1088.901,171.777,430.230,175.780,20.201,153.129
C00641=1088.908,172.027,430.209,175.783,20.202,153.129
C00642=1088.913,172.275,430.186,175.785,20.203,153.129
C00643=1088.919,172.524,430.164,175.788,20.205,153.128
C00644=1088.924,172.773,430.142,175.790,20.206,153.128
C00645=1088.930,173.022,430.121,175.793,20.207,153.128
C00646=1088.935,173.271,430.099,175.796,20.209,153.128
C00647=1088.941,173.520,430.076,175.798,20.210,153.128
C00648=1088.947,173.769,430.055,175.801,20.211,153.128
C00649=1088.952,174.018,430.032,175.803,20.213,153.127
C00650=1088.958,174.267,430.011,175.806,20.214,153.127
C00651=1088.963,174.516,429.988,175.809,20.215,153.127
C00652=1088.969,174.765,429.966,175.812,20.216,153.127
C00653=1088.974,175.014,429.945,175.814,20.218,153.127
C00654=1088.980,175.263,429.922,175.817,20.219,153.127
C00655=1088.986,175.540,429.898,175.820,20.220,153.126
C00656=1088.992,175.817,429.873,175.822,20.222,153.126
C00657=1088.998,176.095,429.848,175.825,20.223,153.126
C00658=1089.005,176.372,429.823,175.828,20.225,153.126
C00659=1089.010,176.621,429.801,175.831,20.226,153.125
C00660=1089.017,176.870,429.779,175.834,20.227,153.125
C00661=1089.022,177.119,429.757,175.836,20.228,153.125
C00662=1089.027,177.368,429.735,175.839,20.230,153.125
C00663=1089.033,177.616,429.713,175.842,20.231,153.125
C00664=1089.039,177.866,429.690,175.844,20.232,153.125
C00665=1089.045,178.115,429.667,175.847,20.234,153.125
C00666=1089.050,178.363,429.646,175.850,20.235,153.124
C00667=1089.056,178.612,429.623,175.852,20.236,153.124
C00668=1089.061,178.862,429.601,175.855,20.237,153.124
C00669=1089.067,179.111,429.579,175.858,20.239,153.124
C00670=1089.073,179.359,429.557,175.860,20.240,153.124
C00671=1089.078,179.609,429.535,175.863,20.241,153.123
C00672=1089.084,179.857,429.512,175.865,20.242,153.123
C00673=1089.090,180.107,429.490,175.868,20.243,153.123
C00674=1089.095,180.355,429.467,175.870,20.244,153.123
C00675=1089.102,180.604,429.445,175.873,20.245,153.123
C00676=1089.107,180.853,429.423,175.876,20.246,153.122
C00677=1089.113,181.102,429.400,175.878,20.247,153.122
C00678=1089.118,181.352,429.378,175.881,20.249,153.122
C00679=1089.124,181.599,429.356,175.884,20.250,153.122
C00680=1089.129,181.849,429.333,175.886,20.251,153.122
C00681=1089.135,182.098,429.310,175.889,20.252,153.121
C00682=1089.142,182.346,429.288,175.892,20.254,153.121
C00683=1089.147,182.596,429.266,175.895,20.255,153.121
C00684=1089.152,182.844,429.243,175.897,20.256,153.121
C00685=1089.158,183.093,429.220,175.901,20.258,153.121
C00686=1089.164,183.342,429.199,175.904,20.259,153.120
C00687=1089.170,183.591,429.176,175.906,20.260,153.120
C00688=1089.175,183.840,429.153,175.909,20.261,153.120
C00689=1089.181,184.090,429.131,175.912,20.262,153.120
C00690=1089.187,184.338,429.108,175.914,20.264,153.120
C00691=1089.193,184.586,429.086,175.917,20.265,153.119
C00692=1089.198,184.836,429.063,175.920,20.266,153.119
C00693=1089.204,185.085,429.041,175.922,20.267,153.119
C00694=1089.209,185.334,429.018,175.925,20.269,153.119
C00695=1089.215,185.583,428.995,175.928,20.270,153.119
C00696=1089.220,185.831,428.973,175.930,20.271,153.119
C00697=1089.226,186.080,428.950,175.933,20.272,153.118
C00698=1089.231,186.329,428.927,175.936,20.274,153.118
C00699=1089.237,186.578,428.904,175.938,20.275,153.118
C00700=1089.243,186.827,428.881,175.941,20.276,153.118
C00701=1089.247,187.076,428.859,175.944,20.278,153.118
C00702=1089.253,187.325,428.836,175.946,20.279,153.117
C00703=1089.258,187.574,428.813,175.949,20.280,153.117
C00704=1089.264,187.823,428.790,175.952,20.281,153.117
C00705=1089.270,188.072,428.767,175.954,20.283,153.117
C00706=1089.275,188.320,428.744,175.957,20.284,153.117
C00707=1089.281,188.569,428.721,175.960,20.285,153.117
C00708=1089.286,188.818,428.699,175.962,20.286,153.116
C00709=1089.291,189.067,428.675,175.965,20.288,153.116
C00710=1089.297,189.316,428.652,175.968,20.289,153.116
C00711=1089.303,189.565,428.630,175.970,20.290,153.116
C00712=1089.308,189.813,428.607,175.974,20.292,153.116
C00713=1089.313,190.062,428.584,175.977,20.293,153.115
C00714=1089.319,190.311,428.561,175.979,20.295,153.115
C00715=1089.324,190.560,428.538,175.982,20.296,153.115
C00716=1089.330,190.809,428.515,175.984,20.297,153.115
C00717=1089.336,191.058,428.492,175.987,20.298,153.115
C00718=1089.341,191.307,428.469,175.990,20.299,153.115
C00719=1089.347,191.584,428.444,175.993,20.301,153.114
C00720=1089.354,191.861,428.418,175.996,20.302,153.114
C00721=1089.359,192.138,428.392,175.999,20.304,153.114
C00722=1089.366,192.415,428.366,176.002,20.305,153.114
C00723=1089.372,192.664,428.343,176.005,20.307,153.114
C00724=1089.377,192.912,428.320,176.008,20.308,153.113
C00725=1089.382,193.161,428.297,176.011,20.309,153.113
C00726=1089.387,193.410,428.274,176.013,20.310,153.113
C00727=1089.393,193.659,428.251,176.016,20.311,153.113
C00728=1089.399,193.908,428.228,176.018,20.313,153.113
C00729=1089.405,194.157,428.205,176.021,20.314,153.112
C00730=1089.410,194.406,428.181,176.024,20.315,153.112
C00731=1089.416,194.654,428.158,176.027,20.316,153.112
C00732=1089.421,194.903,428.135,176.029,20.317,153.112
C00733=1089.427,195.152,428.112,176.033,20.319,153.112
C00734=1089.432,195.401,428.088,176.036,20.320,153.111
C00735=1089.438,195.650,428.065,176.038,20.321,153.111
C00736=1089.444,195.899,428.042,176.041,20.323,153.111
C00737=1089.450,196.148,428.019,176.044,20.324,153.111
C00738=1089.455,196.397,427.995,176.046,20.325,153.111
C00739=1089.460,196.646,427.972,176.049,20.326,153.110
C00740=1089.466,196.894,427.949,176.052,20.327,153.110
C00741=1089.471,197.143,427.925,176.054,20.329,153.110
C00742=1089.477,197.392,427.902,176.058,20.330,153.110
C00743=1089.483,197.641,427.879,176.061,20.331,153.109
C00744=1089.489,197.889,427.855,176.063,20.333,153.109
C00745=1089.494,198.138,427.832,176.066,20.334,153.109
C00746=1089.500,198.387,427.809,176.069,20.335,153.109
C00747=1089.506,198.636,427.785,176.072,20.336,153.109
C00748=1089.511,198.885,427.761,176.074,20.337,153.109
C00749=1089.517,199.134,427.738,176.077,20.338,153.108
C00750=1089.523,199.383,427.715,176.080,20.340,153.108
C00751=1089.528,199.632,427.691,176.083,20.341,153.108
C00752=1089.534,199.880,427.668,176.086,20.342,153.108
C00753=1089.540,200.129,427.645,176.089,20.344,153.107
C00754=1089.545,200.378,427.621,176.092,20.345,153.107
C00755=1089.551,200.627,427.597,176.094,20.346,153.107
C00756=1089.557,200.875,427.574,176.097,20.347,153.107
C00757=1089.562,201.125,427.550,176.100,20.348,153.107
C00758=1089.568,201.374,427.527,176.102,20.349,153.106
C00759=1089.573,201.622,427.503,176.106,20.351,153.106
C00760=1089.579,201.871,427.480,176.109,20.352,153.106
C00761=1089.585,202.119,427.456,176.111,20.353,153.106
C00762=1089.590,202.369,427.432,176.114,20.354,153.105
C00763=1089.597,202.618,427.408,176.117,20.355,153.105
C00764=1089.602,202.867,427.385,176.120,20.357,153.105
C00765=1089.608,203.115,427.361,176.123,20.358,153.105
C00766=1089.613,203.364,427.338,176.126,20.359,153.105
C00767=1089.619,203.613,427.314,176.129,20.361,153.104
C00768=1089.624,203.862,427.291,176.131,20.362,153.104
C00769=1089.629,204.110,427.266,176.134,20.363,153.104
C00770=1089.635,204.359,427.243,176.137,20.364,153.104
C00771=1089.641,204.609,427.219,176.140,20.365,153.104
C00772=1089.647,204.857,427.195,176.143,20.367,153.103
C00773=1089.652,205.106,427.171,176.146,20.368,153.103
C00774=1089.657,205.355,427.147,176.149,20.369,153.103
C00775=1089.663,205.603,427.124,176.151,20.370,153.103
C00776=1089.668,205.852,427.100,176.154,20.371,153.103
C00777=1089.674,206.100,427.076,176.157,20.372,153.102
C00778=1089.680,206.350,427.052,176.160,20.374,153.102
C00779=1089.685,206.599,427.028,176.163,20.375,153.102
C00780=1089.691,206.847,427.005,176.166,20.376,153.102
C00781=1089.696,207.096,426.980,176.168,20.377,153.102
C00782=1089.702,207.344,426.956,176.171,20.379,153.101
C00783=1089.725,208.367,426.858,176.241,20.413,153.097
C00784=1089.734,208.748,426.821,176.245,20.417,153.097
C00785=1089.743,209.129,426.784,176.249,20.420,153.097
C00786=1089.751,209.511,426.746,176.254,20.423,153.097
C00787=1089.760,209.892,426.709,176.257,20.427,153.097
C00788=1089.765,210.141,426.684,176.260,20.429,153.097
C00789=1089.771,210.390,426.660,176.263,20.431,153.097
C00790=1089.776,210.639,426.635,176.266,20.433,153.097
C00791=1089.782,210.887,426.612,176.269,20.435,153.097
C00792=1089.788,211.136,426.586,176.271,20.437,153.097
C00793=1089.794,211.384,426.562,176.274,20.440,153.097
C00794=1089.799,211.633,426.538,176.277,20.442,153.097
C00795=1089.805,211.882,426.513,176.280,20.444,153.097
C00796=1089.810,212.131,426.489,176.282,20.446,153.097
C00797=1089.816,212.379,426.464,176.284,20.448,153.097
C00798=1089.822,212.628,426.439,176.288,20.450,153.097
C00799=1089.827,212.877,426.415,176.290,20.452,153.097
C00800=1089.833,213.126,426.391,176.293,20.454,153.097
C00801=1089.838,213.375,426.366,176.296,20.456,153.097
C00802=1089.844,213.623,426.341,176.299,20.459,153.097
C00803=1089.850,213.872,426.317,176.301,20.461,153.097
C00804=1089.855,214.121,426.291,176.305,20.463,153.097
C00805=1089.860,214.369,426.266,176.307,20.465,153.097
C00806=1089.866,214.618,426.242,176.310,20.468,153.097
C00807=1089.872,214.867,426.218,176.312,20.470,153.097
C00808=1089.877,215.115,426.193,176.316,20.472,153.097
C00809=1089.883,215.364,426.168,176.318,20.474,153.098
C00810=1089.888,215.613,426.144,176.321,20.477,153.098
C00811=1089.895,215.862,426.118,176.324,20.478,153.097
C00812=1089.899,216.111,426.094,176.327,20.481,153.097
C00813=1089.905,216.360,426.069,176.329,20.483,153.097
C00814=1089.911,216.608,426.044,176.332,20.485,153.097
C00815=1089.916,216.856,426.020,176.335,20.487,153.098
C00816=1089.922,217.105,425.994,176.338,20.490,153.098
C00817=1089.927,217.354,425.970,176.340,20.492,153.098
C00818=1089.933,217.603,425.944,176.344,20.494,153.098
C00819=1089.938,217.851,425.920,176.346,20.496,153.098
C00820=1089.944,218.100,425.895,176.349,20.498,153.098
C00821=1089.950,218.349,425.870,176.351,20.500,153.098
C00822=1089.956,218.597,425.845,176.355,20.502,153.098
C00823=1089.961,218.847,425.820,176.357,20.504,153.098
C00824=1089.967,219.095,425.795,176.360,20.507,153.098
C00825=1089.973,219.344,425.770,176.363,20.509,153.098
C00826=1089.978,219.592,425.745,176.366,20.511,153.098
C00827=1089.984,219.841,425.721,176.368,20.513,153.098
C00828=1089.989,220.090,425.695,176.371,20.516,153.098
C00829=1089.995,220.339,425.670,176.374,20.518,153.098
C00830=1090.001,220.588,425.645,176.377,20.520,153.098
C00831=1090.007,220.836,425.620,176.380,20.522,153.098
C00832=1090.012,221.085,425.595,176.383,20.524,153.098
C00833=1090.017,221.333,425.570,176.385,20.526,153.098
C00834=1090.024,221.582,425.545,176.388,20.529,153.098
C00835=1090.030,221.831,425.520,176.391,20.531,153.098
C00836=1090.037,222.216,425.481,176.396,20.534,153.098
C00837=1090.047,222.601,425.442,176.399,20.537,153.098
C00838=1090.055,222.986,425.403,176.404,20.541,153.098
C00839=1090.064,223.371,425.364,176.408,20.544,153.098
C00840=1090.069,223.620,425.338,176.411,20.547,153.098
C00841=1090.075,223.868,425.313,176.414,20.549,153.098
C00842=1090.081,224.117,425.288,176.417,20.551,153.098
C00843=1090.086,224.366,425.262,176.419,20.553,153.098
C00844=1090.092,224.614,425.237,176.422,20.556,153.098
C00845=1090.097,224.863,425.211,176.425,20.558,153.098
C00846=1090.103,225.111,425.186,176.428,20.560,153.098
C00847=1090.108,225.360,425.160,176.430,20.562,153.098
C00848=1090.114,225.610,425.136,176.434,20.564,153.098
C00849=1090.119,225.858,425.110,176.436,20.566,153.098
C00850=1090.125,226.107,425.085,176.439,20.569,153.098
C00851=1090.131,226.356,425.059,176.443,20.571,153.098
C00852=1090.136,226.603,425.034,176.445,20.573,153.098
C00853=1090.142,226.852,425.008,176.448,20.575,153.098
C00854=1090.148,227.101,424.983,176.450,20.577,153.098
C00855=1090.153,227.349,424.957,176.454,20.580,153.098
C00856=1090.159,227.598,424.932,176.456,20.582,153.098
C00857=1090.165,227.847,424.906,176.459,20.584,153.098
C00858=1090.171,228.096,424.880,176.461,20.586,153.098
C00859=1090.176,228.344,424.855,176.465,20.589,153.098
C00860=1090.182,228.593,424.830,176.468,20.591,153.098
C00861=1090.187,228.842,424.804,176.470,20.593,153.098
C00862=1090.194,229.090,424.778,176.474,20.595,153.098
C00863=1090.198,229.339,424.753,176.476,20.597,153.098
C00864=1090.204,229.588,424.727,176.479,20.600,153.098
C00865=1090.210,229.836,424.701,176.482,20.602,153.098
C00866=1090.216,230.085,424.675,176.485,20.604,153.098
C00867=1090.221,230.333,424.651,176.488,20.607,153.098
C00868=1090.227,230.582,424.625,176.490,20.609,153.098
C00869=1090.232,230.831,424.599,176.494,20.611,153.098
C00870=1090.239,231.079,424.573,176.496,20.613,153.098
C00871=1090.244,231.327,424.547,176.499,20.615,153.098
C00872=1090.249,231.576,424.521,176.502,20.618,153.098
C00873=1090.255,231.825,424.496,176.505,20.620,153.098
C00874=1090.261,232.074,424.470,176.508,20.622,153.098
C00875=1090.266,232.323,424.444,176.510,20.624,153.098
C00876=1090.271,232.571,424.418,176.513,20.627,153.098
C00877=1090.278,232.819,424.392,176.516,20.629,153.098
C00878=1090.283,233.068,424.366,176.519,20.631,153.098
C00879=1090.288,233.317,424.340,176.522,20.634,153.099
C00880=1090.294,233.566,424.314,176.525,20.636,153.099
C00881=1090.300,233.814,424.289,176.528,20.638,153.099
C00882=1090.305,234.063,424.263,176.530,20.640,153.099
C00883=1090.311,234.311,424.236,176.533,20.643,153.099
C00884=1090.317,234.560,424.210,176.536,20.645,153.099
C00885=1090.322,234.809,424.184,176.539,20.647,153.099
C00886=1090.328,235.057,424.158,176.542,20.649,153.099
C00887=1090.333,235.305,424.133,176.544,20.651,153.099
C00888=1090.341,235.683,424.093,176.549,20.655,153.099
C00889=1090.350,236.059,424.053,176.553,20.658,153.099
C00890=1090.359,236.435,424.014,176.558,20.662,153.099
C00891=1090.367,236.812,423.974,176.562,20.665,153.099
C00892=1090.372,237.060,423.948,176.565,20.668,153.099
C00893=1090.378,237.309,423.922,176.568,20.670,153.099
C00894=1090.384,237.557,423.896,176.571,20.672,153.099
C00895=1090.390,237.806,423.870,176.574,20.675,153.099
C00896=1090.396,238.054,423.844,176.577,20.677,153.099
C00897=1090.401,238.303,423.818,176.579,20.679,153.099
C00898=1090.407,238.552,423.791,176.583,20.681,153.099
C00899=1090.412,238.801,423.765,176.585,20.683,153.099
C00900=1090.418,239.049,423.738,176.588,20.686,153.099
C00901=1090.424,239.298,423.712,176.591,20.688,153.099
C00902=1090.429,239.546,423.686,176.594,20.690,153.099
C00903=1090.435,239.795,423.659,176.597,20.693,153.099
C00904=1090.441,240.044,423.633,176.600,20.695,153.099
C00905=1090.446,240.291,423.607,176.603,20.697,153.099
C00906=1090.452,240.540,423.580,176.606,20.700,153.099
C00907=1090.457,240.789,423.554,176.609,20.702,153.099
C00908=1090.463,241.037,423.528,176.611,20.704,153.099
C00909=1090.468,241.286,423.502,176.614,20.707,153.099
C00910=1090.474,241.534,423.475,176.617,20.709,153.099
C00911=1090.480,241.783,423.449,176.620,20.711,153.099
C00912=1090.486,242.031,423.422,176.623,20.713,153.099
C00913=1090.491,242.280,423.396,176.626,20.715,153.099
C00914=1090.497,242.529,423.369,176.629,20.718,153.099
C00915=1090.503,242.777,423.343,176.632,20.720,153.099
C00916=1090.508,243.025,423.316,176.634,20.722,153.100
C00917=1090.514,243.274,423.290,176.638,20.725,153.100
C00918=1090.519,243.523,423.263,176.641,20.727,153.100
C00919=1090.525,243.771,423.236,176.643,20.729,153.100
C00920=1090.530,244.020,423.210,176.646,20.732,153.100
C00921=1090.536,244.268,423.183,176.650,20.734,153.100
C00922=1090.542,244.517,423.157,176.652,20.737,153.100
C00923=1090.547,244.765,423.130,176.655,20.739,153.100
C00924=1090.553,245.015,423.103,176.658,20.741,153.100
C00925=1090.559,245.263,423.076,176.660,20.743,153.100
C00926=1090.565,245.511,423.049,176.664,20.746,153.100
C00927=1090.570,245.760,423.023,176.667,20.748,153.100
C00928=1090.575,246.008,422.995,176.669,20.750,153.100
C00929=1090.581,246.257,422.969,176.672,20.753,153.100
C00930=1090.587,246.505,422.942,176.676,20.755,153.100
C00931=1090.592,246.754,422.916,176.678,20.757,153.100
C00932=1090.597,247.003,422.889,176.681,20.760,153.100
C00933=1090.603,247.251,422.862,176.684,20.762,153.100
C00934=1090.609,247.500,422.836,176.687,20.765,153.100
C00935=1090.614,247.748,422.808,176.690,20.767,153.100
C00936=1090.620,247.997,422.782,176.693,20.769,153.100
C00937=1090.626,248.245,422.755,176.696,20.772,153.100
C00938=1090.631,248.493,422.727,176.699,20.774,153.100
C00939=1090.637,248.741,422.701,176.702,20.777,153.101
C00940=1090.645,249.112,422.660,176.706,20.780,153.101
C00941=1090.653,249.481,422.621,176.710,20.784,153.101
C00942=1090.662,249.851,422.580,176.715,20.788,153.101
C00943=1090.670,250.220,422.540,176.719,20.791,153.101
C00944=1090.675,250.469,422.513,176.722,20.794,153.101
C00945=1090.681,250.718,422.486,176.725,20.796,153.101
C00946=1090.686,250.966,422.458,176.728,20.798,153.101
C00947=1090.692,251.214,422.431,176.731,20.800,153.101
C00948=1090.697,251.463,422.404,176.734,20.803,153.101
C00949=1090.703,251.711,422.377,176.736,20.805,153.101
C00950=1090.708,251.960,422.350,176.739,20.808,153.101
C00951=1090.714,252.208,422.323,176.743,20.810,153.101
C00952=1090.720,252.457,422.295,176.746,20.813,153.101
C00953=1090.725,252.705,422.269,176.748,20.815,153.101
C00954=1090.731,252.954,422.241,176.751,20.818,153.101
C00955=1090.737,253.202,422.214,176.754,20.820,153.102
C00956=1090.742,253.450,422.187,176.757,20.822,153.102
C00957=1090.748,253.700,422.160,176.760,20.824,153.102
C00958=1090.753,253.948,422.132,176.763,20.827,153.102
C00959=1090.759,254.196,422.105,176.766,20.829,153.102
C00960=1090.764,254.445,422.078,176.769,20.832,153.102
C00961=1090.770,254.692,422.050,176.772,20.834,153.102
C00962=1090.776,254.942,422.023,176.775,20.837,153.102
C00963=1090.782,255.189,421.995,176.778,20.839,153.102
C00964=1090.787,255.438,421.968,176.781,20.841,153.102
C00965=1090.792,255.686,421.940,176.784,20.844,153.102
C00966=1090.799,255.935,421.913,176.787,20.847,153.102
C00967=1090.804,256.184,421.886,176.790,20.849,153.102
C00968=1090.810,256.432,421.859,176.792,20.851,153.102
C00969=1090.815,256.680,421.831,176.796,20.853,153.102
C00970=1090.821,256.929,421.803,176.799,20.856,153.102
C00971=1090.827,257.177,421.776,176.802,20.858,153.102
C00972=1090.832,257.425,421.748,176.804,20.861,153.102
C00973=1090.839,257.674,421.721,176.807,20.863,153.102
C00974=1090.844,257.923,421.694,176.811,20.866,153.102
C00975=1090.849,258.171,421.666,176.814,20.868,153.103
C00976=1090.855,258.420,421.639,176.816,20.870,153.103
C00977=1090.861,258.668,421.611,176.819,20.873,153.103
C00978=1090.867,258.915,421.583,176.822,20.875,153.103
C00979=1090.872,259.165,421.556,176.826,20.878,153.103
C00980=1090.878,259.413,421.528,176.828,20.880,153.103
C00981=1090.884,259.661,421.501,176.831,20.882,153.103
C00982=1090.889,259.910,421.473,176.834,20.885,153.103
C00983=1090.895,260.158,421.445,176.838,20.887,153.103
C00984=1090.901,260.407,421.418,176.840,20.889,153.103
C00985=1090.907,260.655,421.390,176.843,20.892,153.103
C00986=1090.912,260.903,421.362,176.846,20.895,153.103
C00987=1090.919,261.152,421.334,176.849,20.897,153.103
C00988=1090.924,261.400,421.307,176.853,20.899,153.103
C00989=1090.930,261.649,421.278,176.855,20.901,153.103
C00990=1090.935,261.897,421.251,176.858,20.904,153.103
C00991=1090.941,262.145,421.223,176.861,20.907,153.103
C00992=1090.950,262.512,421.182,176.866,20.910,153.103
C00993=1090.958,262.879,421.141,176.870,20.914,153.104
C00994=1090.967,263.245,421.099,176.875,20.918,153.104
C00995=1090.975,263.612,421.058,176.879,20.921,153.104
C00996=1090.981,263.861,421.031,176.882,20.923,153.104
C00997=1090.987,264.109,421.003,176.885,20.926,153.104
C00998=1090.993,264.358,420.975,176.888,20.928,153.104
C00999=1090.998,264.606,420.947,176.891,20.930,153.104
C01000=1091.003,264.854,420.919,176.894,20.933,153.104
C01001=1091.009,265.103,420.891,176.897,20.936,153.104
C01002=1091.015,265.351,420.863,176.900,20.938,153.104
C01003=1091.021,265.599,420.834,176.903,20.941,153.104
C01004=1091.026,265.847,420.807,176.905,20.943,153.104
C01005=1091.032,266.096,420.778,176.909,20.945,153.104
C01006=1091.037,266.344,420.750,176.912,20.948,153.104
C01007=1091.043,266.593,420.722,176.915,20.951,153.105
C01008=1091.049,266.841,420.694,176.918,20.953,153.105
C01009=1091.055,267.090,420.666,176.921,20.956,153.105
C01010=1091.060,267.338,420.638,176.923,20.958,153.105
C01011=1091.065,267.586,420.610,176.927,20.961,153.105
C01012=1091.071,267.835,420.581,176.930,20.963,153.105
C01013=1091.077,268.082,420.553,176.933,20.966,153.105
C01014=1091.083,268.331,420.524,176.936,20.968,153.105
C01015=1091.089,268.580,420.496,176.939,20.971,153.105
C01016=1091.094,268.828,420.468,176.941,20.973,153.105
C01017=1091.100,269.076,420.440,176.945,20.976,153.105
C01018=1091.105,269.324,420.412,176.948,20.978,153.105
C01019=1091.112,269.573,420.383,176.951,20.981,153.105
C01020=1091.117,269.821,420.355,176.954,20.984,153.106
C01021=1091.123,270.069,420.326,176.957,20.986,153.106
C01022=1091.127,270.318,420.298,176.960,20.988,153.106
C01023=1091.134,270.566,420.269,176.963,20.991,153.106
C01024=1091.139,270.814,420.241,176.966,20.994,153.106
C01025=1091.145,271.063,420.213,176.969,20.996,153.106
C01026=1091.150,271.311,420.185,176.972,20.999,153.106
C01027=1091.157,271.559,420.156,176.975,21.002,153.106
C01028=1091.162,271.808,420.127,176.978,21.004,153.106
C01029=1091.167,272.056,420.099,176.981,21.007,153.106
C01030=1091.173,272.304,420.070,176.984,21.009,153.106
C01031=1091.179,272.552,420.042,176.987,21.011,153.106
C01032=1091.185,272.800,420.013,176.990,21.014,153.107
C01033=1091.190,273.049,419.984,176.993,21.017,153.107
C01034=1091.196,273.297,419.956,176.996,21.020,153.107
C01035=1091.202,273.545,419.927,176.999,21.022,153.107
C01036=1091.207,273.794,419.899,177.002,21.024,153.107
C01037=1091.213,274.042,419.870,177.005,21.027,153.107
C01038=1091.219,274.291,419.841,177.008,21.029,153.107
C01039=1091.224,274.538,419.812,177.011,21.032,153.107
C01040=1091.230,274.787,419.784,177.014,21.035,153.107
C01041=1091.235,275.035,419.755,177.017,21.038,153.107
C01042=1091.241,275.283,419.726,177.020,21.040,153.108
C01043=1091.247,275.532,419.697,177.023,21.043,153.108
C01044=1091.255,275.901,419.655,177.027,21.047,153.108
C01045=1091.264,276.270,419.611,177.032,21.050,153.108
C01046=1091.272,276.640,419.569,177.037,21.054,153.108
C01047=1091.281,277.009,419.525,177.041,21.058,153.108
C01048=1091.285,277.258,419.497,177.044,21.061,153.108
C01049=1091.292,277.506,419.468,177.047,21.064,153.109
C01050=1091.298,277.755,419.439,177.050,21.066,153.109
C01051=1091.303,278.003,419.410,177.053,21.069,153.109
C01052=1091.309,278.250,419.381,177.056,21.071,153.109
C01053=1091.314,278.499,419.351,177.059,21.074,153.109
C01054=1091.320,278.748,419.323,177.062,21.077,153.109
C01055=1091.325,278.995,419.294,177.065,21.080,153.109
C01056=1091.331,279.244,419.265,177.068,21.082,153.109
C01057=1091.338,279.492,419.236,177.071,21.085,153.109
C01058=1091.343,279.741,419.207,177.074,21.087,153.110
C01059=1091.349,279.988,419.178,177.077,21.090,153.110
C01060=1091.354,280.237,419.149,177.080,21.093,153.110
C01061=1091.360,280.485,419.120,177.083,21.095,153.110
C01062=1091.366,280.733,419.090,177.086,21.098,153.110
C01063=1091.371,280.981,419.062,177.090,21.101,153.110
C01064=1091.377,281.230,419.032,177.093,21.104,153.110
C01065=1091.383,281.478,419.003,177.096,21.106,153.110
C01066=1091.388,281.726,418.974,177.099,21.109,153.110
C01067=1091.393,281.974,418.944,177.102,21.112,153.111
C01068=1091.400,282.222,418.915,177.104,21.114,153.111
C01069=1091.405,282.471,418.886,177.107,21.117,153.111
C01070=1091.411,282.719,418.856,177.110,21.120,153.111
C01071=1091.416,282.966,418.827,177.113,21.122,153.111
C01072=1091.422,283.215,418.798,177.117,21.125,153.111
C01073=1091.427,283.463,418.768,177.120,21.128,153.111
C01074=1091.434,283.711,418.739,177.123,21.131,153.111
C01075=1091.439,283.960,418.709,177.126,21.133,153.112
C01076=1091.444,284.208,418.680,177.129,21.136,153.112
C01077=1091.450,284.456,418.651,177.132,21.139,153.112
C01078=1091.456,284.704,418.621,177.135,21.141,153.112
C01079=1091.461,284.953,418.592,177.138,21.144,153.112
C01080=1091.467,285.201,418.563,177.141,21.147,153.112
C01081=1091.472,285.448,418.534,177.144,21.150,153.112
C01082=1091.478,285.697,418.504,177.147,21.153,153.112
C01083=1091.484,285.945,418.475,177.149,21.155,153.113
C01084=1091.490,286.193,418.445,177.153,21.158,153.113
C01085=1091.495,286.441,418.415,177.156,21.160,153.113
C01086=1091.501,286.690,418.385,177.159,21.163,153.113
C01087=1091.507,286.938,418.356,177.162,21.166,153.113
C01088=1091.512,287.186,418.327,177.165,21.169,153.113
C01089=1091.518,287.433,418.297,177.168,21.172,153.113
C01090=1091.523,287.682,418.267,177.171,21.174,153.114
C01091=1091.530,287.930,418.238,177.174,21.177,153.114
C01092=1091.535,288.178,418.208,177.177,21.180,153.114
C01093=1091.541,288.426,418.178,177.180,21.183,153.114
C01094=1091.547,288.675,418.148,177.183,21.186,153.114
C01095=1091.553,288.923,418.119,177.187,21.188,153.114
C01096=1091.561,289.301,418.073,177.191,21.192,153.114
C01097=1091.570,289.681,418.028,177.196,21.197,153.115
C01098=1091.579,290.059,417.982,177.200,21.201,153.115
C01099=1091.588,290.438,417.937,177.205,21.205,153.115
C01100=1091.593,290.687,417.908,177.208,21.208,153.115
C01101=1091.599,290.934,417.877,177.211,21.211,153.115
C01102=1091.604,291.183,417.848,177.214,21.214,153.116
C01103=1091.610,291.431,417.817,177.217,21.217,153.116
C01104=1091.616,291.679,417.788,177.220,21.219,153.116
C01105=1091.621,291.927,417.757,177.223,21.222,153.116
C01106=1091.627,292.175,417.728,177.226,21.225,153.116
C01107=1091.633,292.423,417.697,177.229,21.228,153.116
C01108=1091.638,292.672,417.668,177.232,21.231,153.117
C01109=1091.644,292.919,417.637,177.235,21.234,153.117
C01110=1091.650,293.168,417.608,177.238,21.237,153.117
C01111=1091.655,293.416,417.577,177.241,21.239,153.117
C01112=1091.661,293.664,417.547,177.244,21.242,153.117
C01113=1091.667,293.912,417.517,177.248,21.245,153.117
C01114=1091.673,294.160,417.487,177.251,21.248,153.117
C01115=1091.678,294.408,417.457,177.254,21.251,153.118
C01116=1091.684,294.656,417.427,177.257,21.253,153.118
C01117=1091.690,294.904,417.397,177.260,21.256,153.118
C01118=1091.695,295.152,417.367,177.263,21.259,153.118
C01119=1091.701,295.400,417.337,177.266,21.262,153.118
C01120=1091.707,295.648,417.306,177.269,21.265,153.119
C01121=1091.712,295.896,417.277,177.272,21.268,153.119
C01122=1091.718,296.145,417.246,177.275,21.271,153.119
C01123=1091.723,296.392,417.215,177.279,21.274,153.119
C01124=1091.729,296.640,417.185,177.282,21.277,153.119
C01125=1091.735,296.888,417.155,177.285,21.280,153.119
C01126=1091.741,297.137,417.125,177.288,21.283,153.120
C01127=1091.747,297.385,417.094,177.291,21.286,153.120
C01128=1091.753,297.633,417.064,177.294,21.289,153.120
C01129=1091.758,297.881,417.033,177.297,21.292,153.120
C01130=1091.764,298.129,417.003,177.300,21.295,153.120
C01131=1091.769,298.377,416.973,177.303,21.297,153.120
C01132=1091.775,298.625,416.943,177.306,21.300,153.121
C01133=1091.780,298.873,416.912,177.309,21.303,153.121
C01134=1091.786,299.121,416.881,177.312,21.307,153.121
C01135=1091.791,299.369,416.851,177.315,21.310,153.121
C01136=1091.797,299.617,416.820,177.318,21.312,153.122
C01137=1091.803,299.865,416.790,177.321,21.315,153.122
C01138=1091.808,300.113,416.759,177.324,21.318,153.122
C01139=1091.814,300.361,416.728,177.327,21.322,153.122
C01140=1091.820,300.609,416.698,177.330,21.324,153.122
C01141=1091.825,300.857,416.667,177.334,21.328,153.123
C01142=1091.831,301.105,416.637,177.337,21.331,153.123
C01143=1091.836,301.353,416.606,177.340,21.334,153.123
C01144=1091.842,301.601,416.575,177.343,21.337,153.123
C01145=1091.847,301.849,416.544,177.346,21.340,153.123
C01146=1091.853,302.097,416.514,177.349,21.343,153.124
C01147=1091.859,302.346,416.483,177.351,21.346,153.124
C01148=1091.867,302.738,416.435,177.357,21.351,153.124
C01149=1091.876,303.131,416.386,177.361,21.356,153.125
C01150=1091.885,303.524,416.336,177.366,21.360,153.125
C01151=1091.894,303.917,416.288,177.371,21.365,153.125
C01152=1091.900,304.165,416.257,177.374,21.368,153.125
C01153=1091.905,304.412,416.227,177.377,21.371,153.126
C01154=1091.911,304.661,416.195,177.380,21.375,153.126
C01155=1091.917,304.909,416.164,177.383,21.377,153.126
C01156=1091.922,305.157,416.133,177.387,21.381,153.126
C01157=1091.928,305.404,416.103,177.390,21.384,153.127
C01158=1091.934,305.653,416.071,177.393,21.387,153.127
C01159=1091.940,305.900,416.040,177.396,21.390,153.127
C01160=1091.945,306.149,416.010,177.399,21.393,153.127
C01161=1091.951,306.396,415.978,177.402,21.396,153.127
C01162=1091.957,306.645,415.947,177.405,21.399,153.128
C01163=1091.963,306.892,415.917,177.407,21.403,153.128
C01164=1091.968,307.140,415.885,177.411,21.406,153.128
C01165=1091.973,307.388,415.854,177.414,21.409,153.128
C01166=1091.979,307.637,415.823,177.417,21.412,153.129
C01167=1091.985,307.884,415.792,177.420,21.415,153.129
C01168=1091.991,308.132,415.761,177.423,21.418,153.129
C01169=1091.997,308.380,415.729,177.426,21.421,153.129
C01170=1092.002,308.628,415.699,177.429,21.424,153.129
C01171=1092.008,308.876,415.667,177.432,21.427,153.130
C01172=1092.014,309.124,415.636,177.436,21.431,153.130
C01173=1092.020,309.372,415.605,177.439,21.434,153.130
C01174=1092.025,309.620,415.574,177.442,21.437,153.130
C01175=1092.031,309.868,415.543,177.445,21.440,153.131
C01176=1092.037,310.116,415.512,177.448,21.443,153.131
C01177=1092.043,310.364,415.480,177.451,21.446,153.131
C01178=1092.049,310.611,415.449,177.454,21.449,153.131
C01179=1092.054,310.860,415.417,177.457,21.453,153.132
C01180=1092.060,311.107,415.386,177.460,21.456,153.132
C01181=1092.066,311.355,415.355,177.463,21.459,153.132
C01182=1092.072,311.604,415.323,177.466,21.462,153.132
C01183=1092.077,311.851,415.292,177.469,21.465,153.133
C01184=1092.083,312.100,415.261,177.472,21.468,153.133
C01185=1092.089,312.347,415.229,177.476,21.472,153.133
C01186=1092.095,312.595,415.197,177.479,21.475,153.133
C01187=1092.101,312.842,415.166,177.482,21.478,153.133
C01188=1092.106,313.091,415.135,177.485,21.481,153.134
C01189=1092.112,313.339,415.103,177.488,21.484,153.134
C01190=1092.119,313.587,415.072,177.491,21.487,153.134
C01191=1092.124,313.834,415.040,177.495,21.491,153.134
C01192=1092.130,314.083,415.009,177.498,21.494,153.135
C01193=1092.136,314.330,414.978,177.500,21.497,153.135
C01194=1092.142,314.579,414.946,177.503,21.500,153.135
C01195=1092.147,314.826,414.914,177.506,21.503,153.136
C01196=1092.153,315.074,414.882,177.509,21.506,153.136
C01197=1092.159,315.322,414.850,177.513,21.510,153.136
C01198=1092.164,315.571,414.819,177.516,21.513,153.136
C01199=1092.170,315.818,414.787,177.519,21.517,153.137
C01200=1092.179,316.214,414.737,177.524,21.522,153.137
C01201=1092.188,316.609,414.686,177.528,21.527,153.138
C01202=1092.197,317.005,414.635,177.533,21.533,153.138
C01203=1092.205,317.400,414.584,177.538,21.538,153.139
C01204=1092.211,317.648,414.552,177.541,21.542,153.139
C01205=1092.217,317.896,414.520,177.544,21.545,153.139
C01206=1092.223,318.144,414.488,177.547,21.548,153.140
C01207=1092.228,318.391,414.456,177.551,21.552,153.140
C01208=1092.234,318.640,414.424,177.553,21.556,153.140
C01209=1092.239,318.888,414.392,177.556,21.558,153.140
C01210=1092.245,319.136,414.360,177.559,21.562,153.141
C01211=1092.251,319.384,414.328,177.562,21.565,153.141
C01212=1092.256,319.631,414.297,177.566,21.569,153.141
C01213=1092.262,319.879,414.264,177.569,21.572,153.142
C01214=1092.268,320.126,414.232,177.572,21.576,153.142
C01215=1092.273,320.375,414.199,177.574,21.579,153.142
C01216=1092.279,320.623,414.167,177.578,21.583,153.143
C01217=1092.284,320.871,414.136,177.581,21.586,153.143
C01218=1092.290,321.119,414.104,177.584,21.589,153.143
C01219=1092.296,321.366,414.071,177.587,21.593,153.144
C01220=1092.302,321.614,414.039,177.590,21.597,153.144
C01221=1092.307,321.863,414.007,177.593,21.600,153.144
C01222=1092.313,322.110,413.975,177.596,21.603,153.145
C01223=1092.319,322.358,413.942,177.599,21.607,153.145
C01224=1092.325,322.606,413.910,177.603,21.610,153.145
C01225=1092.330,322.854,413.878,177.605,21.614,153.145
C01226=1092.336,323.101,413.845,177.608,21.617,153.146
C01227=1092.342,323.350,413.813,177.611,21.620,153.146
C01228=1092.347,323.597,413.782,177.615,21.624,153.146
C01229=1092.353,323.845,413.748,177.618,21.628,153.147
C01230=1092.359,324.093,413.716,177.621,21.631,153.147
C01231=1092.365,324.340,413.684,177.623,21.634,153.147
C01232=1092.371,324.588,413.652,177.627,21.639,153.148
C01233=1092.376,324.837,413.619,177.630,21.642,153.148
C01234=1092.382,325.084,413.586,177.633,21.645,153.149
C01235=1092.388,325.332,413.555,177.636,21.649,153.149
C01236=1092.394,325.580,413.522,177.639,21.652,153.149
C01237=1092.399,325.828,413.489,177.642,21.656,153.149
C01238=1092.405,326.076,413.457,177.645,21.659,153.150
C01239=1092.411,326.323,413.425,177.649,21.663,153.150
C01240=1092.416,326.571,413.392,177.651,21.666,153.150
C01241=1092.422,326.819,413.360,177.654,21.670,153.151
C01242=1092.429,327.067,413.327,177.658,21.674,153.151
C01243=1092.434,327.315,413.294,177.661,21.677,153.152
C01244=1092.440,327.562,413.262,177.664,21.681,153.152
C01245=1092.446,327.810,413.229,177.666,21.684,153.152
C01246=1092.451,328.058,413.196,177.670,21.688,153.153
C01247=1092.457,328.306,413.164,177.673,21.691,153.153
C01248=1092.464,328.554,413.131,177.676,21.695,153.153
C01249=1092.469,328.801,413.098,177.679,21.699,153.154
C01250=1092.475,329.050,413.066,177.682,21.702,153.154
C01251=1092.480,329.297,413.033,177.685,21.706,153.154
C01252=1092.490,329.685,412.981,177.690,21.711,153.155
C01253=1092.498,330.075,412.930,177.695,21.717,153.155
C01254=1092.508,330.463,412.879,177.700,21.723,153.156
C01255=1092.517,330.852,412.827,177.705,21.729,153.157
C01256=1092.523,331.099,412.794,177.708,21.732,153.157
C01257=1092.529,331.347,412.761,177.711,21.736,153.157
C01258=1092.535,331.595,412.729,177.714,21.739,153.158
C01259=1092.541,331.843,412.696,177.717,21.743,153.158
C01260=1092.547,332.091,412.663,177.720,21.747,153.158
C01261=1092.552,332.339,412.630,177.723,21.751,153.159
C01262=1092.558,332.586,412.597,177.726,21.754,153.159
C01263=1092.564,332.834,412.563,177.729,21.758,153.160
C01264=1092.570,333.082,412.530,177.733,21.762,153.160
C01265=1092.575,333.329,412.498,177.735,21.766,153.161
C01266=1092.581,333.577,412.464,177.738,21.769,153.161
C01267=1092.586,333.825,412.431,177.742,21.773,153.161
C01268=1092.593,334.072,412.398,177.744,21.777,153.162
C01269=1092.598,334.320,412.365,177.748,21.781,153.162
C01270=1092.604,334.568,412.332,177.751,21.784,153.163
C01271=1092.609,334.816,412.298,177.753,21.788,153.163
C01272=1092.616,335.064,412.266,177.757,21.792,153.163
C01273=1092.621,335.312,412.232,177.760,21.796,153.164
C01274=1092.627,335.559,412.199,177.763,21.800,153.164
C01275=1092.633,335.806,412.165,177.766,21.804,153.165
C01276=1092.639,336.054,412.132,177.769,21.807,153.165
C01277=1092.644,336.302,412.099,177.772,21.811,153.165
C01278=1092.650,336.550,412.065,177.775,21.815,153.166
C01279=1092.656,336.798,412.032,177.779,21.820,153.166
C01280=1092.662,337.046,411.999,177.781,21.823,153.167
C01281=1092.668,337.293,411.965,177.784,21.827,153.167
C01282=1092.673,337.541,411.932,177.788,21.831,153.168
C01283=1092.679,337.789,411.899,177.790,21.835,153.168
C01284=1092.685,338.036,411.866,177.794,21.838,153.168
C01285=1092.691,338.284,411.832,177.797,21.842,153.169
C01286=1092.697,338.531,411.798,177.800,21.846,153.169
C01287=1092.702,338.779,411.765,177.803,21.850,153.170
C01288=1092.708,339.027,411.731,177.806,21.854,153.170
C01289=1092.714,339.275,411.698,177.809,21.858,153.171
C01290=1092.719,339.522,411.664,177.812,21.862,153.171
C01291=1092.725,339.770,411.630,177.815,21.866,153.172
C01292=1092.730,340.018,411.597,177.818,21.870,153.172
C01293=1092.736,340.265,411.563,177.821,21.874,153.173
C01294=1092.743,340.514,411.529,177.824,21.878,153.173
C01295=1092.748,340.761,411.496,177.828,21.882,153.174
C01296=1092.754,341.009,411.462,177.830,21.886,153.174
C01297=1092.759,341.257,411.429,177.834,21.890,153.174
C01298=1092.765,341.504,411.394,177.837,21.894,153.175
C01299=1092.771,341.752,411.361,177.840,21.899,153.176
C01300=1092.777,341.999,411.327,177.843,21.903,153.176
C01301=1092.782,342.247,411.294,177.845,21.906,153.176
C01302=1092.788,342.494,411.260,177.849,21.911,153.177
C01303=1092.795,342.742,411.225,177.851,21.914,153.177
C01304=1092.803,343.124,411.174,177.856,21.921,153.178
C01305=1092.812,343.507,411.121,177.861,21.927,153.179
C01306=1092.821,343.890,411.069,177.866,21.934,153.180
C01307=1092.830,344.273,411.017,177.871,21.940,153.180
C01308=1092.837,344.521,410.982,177.874,21.944,153.181
C01309=1092.842,344.768,410.949,177.877,21.948,153.181
C01310=1092.847,345.016,410.914,177.880,21.953,153.182
C01311=1092.853,345.263,410.880,177.883,21.956,153.182
C01312=1092.859,345.511,410.846,177.886,21.961,153.183
C01313=1092.865,345.759,410.812,177.889,21.965,153.183
C01314=1092.871,346.007,410.778,177.892,21.969,153.184
C01315=1092.876,346.254,410.744,177.895,21.973,153.185
C01316=1092.882,346.501,410.710,177.899,21.978,153.185
C01317=1092.888,346.749,410.676,177.901,21.982,153.186
C01318=1092.894,346.997,410.641,177.905,21.986,153.186
C01319=1092.899,347.245,410.607,177.908,21.991,153.187
C01320=1092.905,347.492,410.573,177.911,21.994,153.187
C01321=1092.911,347.739,410.539,177.914,21.999,153.188
C01322=1092.917,347.987,410.505,177.917,22.003,153.188
C01323=1092.923,348.235,410.470,177.920,22.008,153.189
C01324=1092.928,348.482,410.436,177.922,22.012,153.189
C01325=1092.934,348.730,410.402,177.926,22.016,153.190
C01326=1092.940,348.978,410.367,177.929,22.020,153.190
C01327=1092.946,349.225,410.333,177.932,22.025,153.191
C01328=1092.952,349.472,410.299,177.935,22.029,153.191
C01329=1092.957,349.720,410.264,177.938,22.033,153.192
C01330=1092.963,349.968,410.230,177.941,22.038,153.193
C01331=1092.969,350.215,410.196,177.944,22.042,153.193
C01332=1092.974,350.463,410.161,177.947,22.047,153.194
C01333=1092.981,350.710,410.126,177.950,22.051,153.194
C01334=1092.986,350.958,410.091,177.953,22.055,153.195
C01335=1092.992,351.205,410.057,177.957,22.060,153.195
C01336=1092.998,351.453,410.023,177.959,22.064,153.196
C01337=1093.004,351.701,409.988,177.963,22.069,153.197
C01338=1093.009,351.948,409.954,177.965,22.073,153.197
C01339=1093.015,352.196,409.918,177.968,22.077,153.198
C01340=1093.021,352.443,409.884,177.972,22.082,153.198
C01341=1093.027,352.690,409.850,177.975,22.086,153.199
C01342=1093.033,352.939,409.815,177.978,22.091,153.199
C01343=1093.039,353.185,409.780,177.980,22.095,153.200
C01344=1093.045,353.434,409.745,177.984,22.099,153.201
C01345=1093.051,353.681,409.711,177.987,22.104,153.201
C01346=1093.056,353.928,409.676,177.990,22.108,153.202
C01347=1093.062,354.176,409.641,177.993,22.113,153.202
C01348=1093.068,354.423,409.607,177.996,22.118,153.203
C01349=1093.073,354.670,409.572,177.999,22.122,153.204
C01350=1093.080,354.918,409.537,178.002,22.127,153.204
C01351=1093.085,355.165,409.502,178.005,22.131,153.205
C01352=1093.091,355.414,409.467,178.008,22.136,153.206
C01353=1093.097,355.661,409.433,178.011,22.141,153.206
C01354=1093.102,355.908,409.397,178.014,22.145,153.207
C01355=1093.108,356.156,409.363,178.017,22.149,153.207
C01356=1093.117,356.541,409.308,178.022,22.157,153.209
C01357=1093.126,356.926,409.254,178.027,22.164,153.209
C01358=1093.135,357.312,409.199,178.032,22.171,153.210
C01359=1093.144,357.696,409.144,178.036,22.178,153.211
C01360=1093.150,357.944,409.109,178.039,22.184,153.212
C01361=1093.156,358.191,409.074,178.042,22.188,153.213
C01362=1093.162,358.439,409.039,178.045,22.192,153.213
C01363=1093.167,358.686,409.004,178.048,22.197,153.214
C01364=1093.174,358.934,408.969,178.052,22.202,153.215
C01365=1093.179,359.181,408.934,178.054,22.207,153.215
C01366=1093.185,359.429,408.899,178.057,22.211,153.216
C01367=1093.191,359.676,408.863,178.061,22.216,153.217
C01368=1093.197,359.923,408.828,178.063,22.221,153.217
C01369=1093.203,360.171,408.793,178.067,22.225,153.218
C01370=1093.209,360.419,408.758,178.070,22.231,153.219
C01371=1093.214,360.666,408.722,178.072,22.235,153.219
C01372=1093.220,360.913,408.687,178.075,22.240,153.220
C01373=1093.226,361.160,408.652,178.079,22.245,153.221
C01374=1093.232,361.408,408.616,178.082,22.250,153.222
C01375=1093.238,361.656,408.581,178.084,22.254,153.222
C01376=1093.243,361.903,408.546,178.088,22.259,153.223
C01377=1093.249,362.151,408.510,178.091,22.265,153.224
C01378=1093.255,362.398,408.475,178.094,22.270,153.224
C01379=1093.261,362.645,408.439,178.097,22.274,153.225
C01380=1093.266,362.892,408.404,178.100,22.279,153.226
C01381=1093.273,363.140,408.368,178.103,22.284,153.226
C01382=1093.279,363.387,408.333,178.105,22.289,153.227
C01383=1093.285,363.634,408.297,178.108,22.294,153.228
C01384=1093.291,363.882,408.262,178.112,22.299,153.229
C01385=1093.296,364.129,408.226,178.115,22.304,153.229
C01386=1093.302,364.377,408.190,178.118,22.309,153.230
C01387=1093.308,364.624,408.155,178.121,22.313,153.231
C01388=1093.314,364.871,408.119,178.124,22.318,153.231
C01389=1093.320,365.118,408.083,178.127,22.324,153.232
C01390=1093.326,365.366,408.047,178.130,22.329,153.233
C01391=1093.331,365.613,408.012,178.133,22.333,153.234
C01392=1093.337,365.861,407.976,178.136,22.339,153.235
C01393=1093.343,366.108,407.940,178.139,22.344,153.235
C01394=1093.349,366.355,407.905,178.142,22.349,153.236
C01395=1093.355,366.602,407.869,178.145,22.354,153.237
C01396=1093.360,366.850,407.832,178.147,22.359,153.238
C01397=1093.366,367.097,407.797,178.151,22.364,153.238
C01398=1093.372,367.345,407.761,178.154,22.369,153.239
C01399=1093.378,367.592,407.725,178.157,22.375,153.240
C01400=1093.384,367.839,407.689,178.160,22.380,153.241
C01401=1093.390,368.087,407.654,178.162,22.385,153.241
C01402=1093.395,368.334,407.617,178.165,22.390,153.242
C01403=1093.401,368.581,407.581,178.169,22.395,153.243
C01404=1093.407,368.828,407.545,178.172,22.400,153.244
C01405=1093.413,369.076,407.509,178.175,22.406,153.245
C01406=1093.419,369.323,407.474,178.178,22.411,153.245
C01407=1093.424,369.570,407.437,178.180,22.416,153.246
C01408=1093.434,369.971,407.379,178.185,22.425,153.248
C01409=1093.443,370.370,407.320,178.190,22.433,153.249
C01410=1093.453,370.772,407.262,178.195,22.442,153.250
C01411=1093.462,371.172,407.202,178.200,22.451,153.252
C01412=1093.468,371.420,407.167,178.203,22.456,153.252
C01413=1093.475,371.667,407.130,178.206,22.461,153.253
C01414=1093.480,371.913,407.094,178.209,22.467,153.254
C01415=1093.486,372.161,407.058,178.212,22.472,153.255
C01416=1093.492,372.408,407.021,178.215,22.477,153.256
C01417=1093.498,372.655,406.985,178.218,22.483,153.257
C01418=1093.504,372.903,406.949,178.221,22.488,153.257
C01419=1093.510,373.150,406.912,178.224,22.494,153.258
C01420=1093.516,373.397,406.876,178.227,22.499,153.259
C01421=1093.521,373.645,406.840,178.230,22.504,153.260
C01422=1093.527,373.892,406.803,178.233,22.509,153.261
C01423=1093.534,374.139,406.767,178.236,22.515,153.262
C01424=1093.539,374.386,406.730,178.239,22.520,153.263
C01425=1093.546,374.633,406.693,178.242,22.526,153.263
C01426=1093.551,374.881,406.657,178.245,22.532,153.264
C01427=1093.557,375.127,406.621,178.248,22.538,153.265
C01428=1093.562,375.375,406.584,178.251,22.543,153.266
C01429=1093.569,375.622,406.548,178.254,22.549,153.267
C01430=1093.574,375.869,406.510,178.257,22.555,153.268
C01431=1093.580,376.116,406.474,178.260,22.560,153.269
C01432=1093.586,376.364,406.437,178.263,22.566,153.270
C01433=1093.592,376.610,406.401,178.266,22.572,153.271
C01434=1093.597,376.857,406.364,178.269,22.577,153.272
C01435=1093.604,377.104,406.327,178.271,22.582,153.273
C01436=1093.609,377.352,406.290,178.274,22.588,153.274
C01437=1093.615,377.599,406.253,178.277,22.594,153.274
C01438=1093.621,377.846,406.217,178.280,22.600,153.275
C01439=1093.627,378.094,406.180,178.283,22.605,153.276
C01440=1093.633,378.341,406.143,178.286,22.611,153.277
C01441=1093.639,378.588,406.106,178.289,22.617,153.278
C01442=1093.644,378.835,406.069,178.292,22.623,153.279
C01443=1093.651,379.082,406.033,178.295,22.628,153.280
C01444=1093.657,379.329,405.995,178.298,22.634,153.281
C01445=1093.663,379.576,405.959,178.300,22.640,153.282
C01446=1093.669,379.824,405.922,178.304,22.646,153.283
C01447=1093.674,380.071,405.885,178.306,22.652,153.284
C01448=1093.680,380.318,405.848,178.309,22.657,153.285
C01449=1093.686,380.565,405.810,178.312,22.663,153.286
C01450=1093.692,380.812,405.773,178.315,22.669,153.287
C01451=1093.698,381.059,405.737,178.318,22.675,153.288
C01452=1093.704,381.306,405.699,178.321,22.681,153.289
C01453=1093.710,381.553,405.662,178.324,22.687,153.290
C01454=1093.716,381.800,405.626,178.327,22.693,153.291
C01455=1093.722,382.047,405.588,178.330,22.699,153.292
C01456=1093.728,382.294,405.551,178.333,22.705,153.293
C01457=1093.734,382.541,405.514,178.336,22.711,153.294
C01458=1093.740,382.788,405.477,178.339,22.717,153.295
C01459=1093.746,383.036,405.440,178.342,22.723,153.296
C01460=1093.755,383.422,405.381,178.346,22.732,153.298
C01461=1093.764,383.807,405.323,178.351,22.742,153.299
C01462=1093.773,384.194,405.264,178.355,22.751,153.301
C01463=1093.782,384.580,405.205,178.360,22.761,153.303
C01464=1093.788,384.827,405.168,178.363,22.767,153.304
C01465=1093.794,385.074,405.131,178.366,22.773,153.305
C01466=1093.800,385.320,405.093,178.369,22.780,153.306
C01467=1093.806,385.568,405.056,178.372,22.786,153.307
C01468=1093.812,385.814,405.018,178.375,22.793,153.308
C01469=1093.818,386.061,404.981,178.378,22.798,153.309
C01470=1093.823,386.309,404.944,178.381,22.805,153.310
C01471=1093.829,386.555,404.906,178.383,22.811,153.311
C01472=1093.836,386.845,404.862,178.387,22.819,153.313
C01473=1093.843,387.133,404.817,178.390,22.826,153.314
C01474=1093.850,387.422,404.774,178.394,22.833,153.315
C01475=1093.857,387.711,404.730,178.397,22.840,153.316
C01476=1093.863,387.958,404.692,178.400,22.847,153.317
C01477=1093.869,388.205,404.655,178.403,22.853,153.319
C01478=1093.875,388.453,404.616,178.406,22.860,153.320
C01479=1093.881,388.699,404.578,178.409,22.866,153.321
C01480=1093.886,388.946,404.540,178.412,22.873,153.322
C01481=1093.892,389.193,404.503,178.414,22.879,153.323
C01482=1093.899,389.440,404.464,178.417,22.886,153.324
C01483=1093.905,389.687,404.427,178.420,22.892,153.325
C01484=1093.911,389.934,404.389,178.424,22.899,153.327
C01485=1093.917,390.180,404.351,178.426,22.905,153.328
C01486=1093.923,390.428,404.313,178.429,22.912,153.329
C01487=1093.929,390.675,404.275,178.432,22.918,153.330
C01488=1093.935,390.921,404.238,178.435,22.924,153.331
C01489=1093.941,391.168,404.200,178.438,22.932,153.332
C01490=1093.947,391.416,404.162,178.441,22.938,153.334
C01491=1093.952,391.663,404.123,178.444,22.944,153.335
C01492=1093.959,391.910,404.085,178.446,22.951,153.336
C01493=1093.965,392.157,404.047,178.449,22.957,153.337
C01494=1093.971,392.404,404.010,178.453,22.965,153.338
C01495=1093.977,392.651,403.972,178.455,22.971,153.340
C01496=1093.983,392.897,403.932,178.458,22.978,153.341
C01497=1093.989,393.144,403.895,178.461,22.984,153.342
C01498=1093.995,393.391,403.857,178.464,22.992,153.343
C01499=1094.000,393.639,403.818,178.467,22.998,153.345
C01500=1094.007,393.885,403.780,178.469,23.005,153.346
C01501=1094.013,394.132,403.742,178.472,23.012,153.347
C01502=1094.018,394.379,403.703,178.476,23.019,153.348
C01503=1094.024,394.625,403.665,178.478,23.026,153.349
C01504=1094.031,394.873,403.627,178.481,23.032,153.351
C01505=1094.036,395.120,403.588,178.483,23.039,153.352
C01506=1094.043,395.367,403.550,178.487,23.046,153.353
C01507=1094.049,395.614,403.512,178.490,23.053,153.355
C01508=1094.054,395.861,403.473,178.492,23.060,153.356
C01509=1094.061,396.107,403.435,178.496,23.067,153.357
C01510=1094.066,396.354,403.396,178.498,23.075,153.359
C01511=1094.073,396.601,403.357,178.501,23.081,153.360
C01512=1094.077,396.821,403.323,178.504,23.088,153.361
C01513=1094.083,397.042,403.288,178.506,23.094,153.362
C01514=1094.088,397.263,403.254,178.508,23.100,153.363
C01515=1094.094,397.483,403.219,178.511,23.107,153.365
C01516=1094.099,397.703,403.185,178.514,23.113,153.366
C01517=1094.105,397.924,403.151,178.516,23.120,153.367
C01518=1094.109,398.144,403.116,178.518,23.126,153.368
C01519=1094.115,398.365,403.081,178.521,23.132,153.369
C01520=1094.121,398.612,403.043,178.524,23.139,153.371
C01521=1094.127,398.859,403.004,178.527,23.147,153.372
C01522=1094.133,399.105,402.965,178.530,23.154,153.373
C01523=1094.139,399.353,402.927,178.533,23.161,153.375
C01524=1094.145,399.600,402.887,178.535,23.169,153.376
C01525=1094.151,399.846,402.849,178.538,23.175,153.377
C01526=1094.157,400.094,402.810,178.541,23.183,153.379
C01527=1094.163,400.340,402.771,178.544,23.190,153.380
C01528=1094.169,400.587,402.732,178.546,23.198,153.382
C01529=1094.175,400.833,402.693,178.550,23.205,153.383
C01530=1094.181,401.081,402.654,178.552,23.213,153.384
C01531=1094.187,401.328,402.615,178.556,23.220,153.386
C01532=1094.193,401.574,402.576,178.558,23.228,153.387
C01533=1094.199,401.822,402.537,178.561,23.236,153.389
C01534=1094.204,402.068,402.498,178.564,23.243,153.390
C01535=1094.211,402.315,402.459,178.566,23.250,153.392
C01536=1094.217,402.562,402.420,178.569,23.258,153.393
C01537=1094.223,402.808,402.381,178.572,23.265,153.395
C01538=1094.229,403.056,402.341,178.575,23.273,153.396
C01539=1094.235,403.303,402.302,178.578,23.281,153.397
C01540=1094.241,403.549,402.263,178.581,23.288,153.399
C01541=1094.247,403.796,402.224,178.583,23.296,153.400
C01542=1094.253,404.043,402.184,178.587,23.304,153.402
C01543=1094.259,404.290,402.145,178.589,23.311,153.403
C01544=1094.265,404.537,402.106,178.592,23.319,153.405
C01545=1094.271,404.784,402.067,178.595,23.327,153.406
C01546=1094.278,405.031,402.028,178.598,23.335,153.408
C01547=1094.284,405.276,401.988,178.600,23.342,153.409
C01548=1094.290,405.524,401.948,178.604,23.350,153.411
C01549=1094.296,405.771,401.909,178.606,23.358,153.412
C01550=1094.302,406.018,401.870,178.609,23.366,153.414
C01551=1094.308,406.264,401.830,178.611,23.374,153.416
C01552=1094.314,406.511,401.790,178.615,23.382,153.417
C01553=1094.320,406.758,401.751,178.618,23.390,153.419
C01554=1094.326,407.005,401.712,178.620,23.398,153.420
C01555=1094.332,407.251,401.672,178.623,23.406,153.422
C01556=1094.338,407.498,401.632,178.626,23.414,153.423
C01557=1094.344,407.745,401.593,178.629,23.422,153.425
C01558=1094.350,407.992,401.553,178.632,23.430,153.427
C01559=1094.356,408.239,401.513,178.634,23.438,153.428
C01560=1094.362,408.485,401.474,178.637,23.447,153.430
C01561=1094.367,408.732,401.433,178.641,23.455,153.431
C01562=1094.374,408.979,401.393,178.643,23.463,153.433
C01563=1094.380,409.226,401.354,178.646,23.472,153.435
C01564=1094.386,409.472,401.314,178.648,23.480,153.436
C01565=1094.392,409.719,401.275,178.651,23.488,153.438
C01566=1094.398,409.965,401.235,178.654,23.496,153.440
C01567=1094.403,410.213,401.195,178.657,23.504,153.441
C01568=1094.409,410.434,401.158,178.660,23.512,153.443
C01569=1094.414,410.654,401.123,178.662,23.520,153.444
C01570=1094.420,410.875,401.087,178.665,23.527,153.446
C01571=1094.425,411.096,401.051,178.667,23.535,153.447
C01572=1094.431,411.317,401.015,178.670,23.543,153.449
C01573=1094.436,411.537,400.979,178.672,23.550,153.450
C01574=1094.441,411.758,400.944,178.674,23.558,153.452
C01575=1094.447,411.979,400.908,178.677,23.565,153.453
C01576=1094.453,412.225,400.868,178.680,23.574,153.455
C01577=1094.459,412.472,400.828,178.683,23.582,153.457
C01578=1094.465,412.719,400.787,178.686,23.591,153.459
C01579=1094.471,412.966,400.748,178.688,23.599,153.460
C01580=1094.477,413.212,400.707,178.691,23.608,153.462
C01581=1094.484,413.459,400.667,178.694,23.617,153.464
C01582=1094.489,413.706,400.627,178.697,23.626,153.465
C01583=1094.496,413.952,400.586,178.700,23.635,153.467
C01584=1094.502,414.199,400.546,178.702,23.643,153.469
C01585=1094.508,414.445,400.506,178.706,23.652,153.471
C01586=1094.514,414.692,400.465,178.709,23.661,153.473
C01587=1094.521,414.938,400.425,178.712,23.670,153.474
C01588=1094.526,415.185,400.385,178.715,23.678,153.476
C01589=1094.533,415.432,400.344,178.718,23.687,153.478
C01590=1094.539,415.678,400.304,178.720,23.696,153.480
C01591=1094.545,415.925,400.263,178.722,23.705,153.482
C01592=1094.551,416.172,400.223,178.725,23.714,153.483
C01593=1094.558,416.419,400.183,178.728,23.723,153.485
C01594=1094.564,416.666,400.142,178.731,23.732,153.487
C01595=1094.570,416.912,400.101,178.734,23.741,153.489
C01596=1094.576,417.158,400.060,178.737,23.751,153.491
C01597=1094.582,417.405,400.020,178.740,23.760,153.493
C01598=1094.588,417.652,399.980,178.743,23.769,153.495
C01599=1094.594,417.898,399.938,178.746,23.778,153.497
C01600=1094.600,418.144,399.898,178.749,23.788,153.498
C01601=1094.606,418.391,399.857,178.751,23.797,153.500
C01602=1094.612,418.638,399.816,178.754,23.806,153.502
C01603=1094.618,418.884,399.776,178.756,23.815,153.504
C01604=1094.624,419.131,399.735,178.759,23.825,153.506
C01605=1094.631,419.377,399.694,178.762,23.834,153.508
C01606=1094.637,419.624,399.653,178.765,23.843,153.510
C01607=1094.643,419.870,399.611,178.768,23.853,153.512
C01608=1094.649,420.117,399.571,178.771,23.862,153.514
C01609=1094.655,420.363,399.530,178.774,23.872,153.516
C01610=1094.661,420.610,399.489,178.776,23.882,153.518
C01611=1094.668,420.857,399.448,178.779,23.891,153.520
C01612=1094.674,421.103,399.407,178.782,23.901,153.522
C01613=1094.680,421.350,399.366,178.786,23.910,153.524
C01614=1094.686,421.596,399.325,178.788,23.920,153.526
C01615=1094.693,421.843,399.284,178.791,23.930,153.528
C01616=1094.699,422.089,399.242,178.794,23.940,153.530
C01617=1094.704,422.335,399.201,178.797,23.949,153.532
C01618=1094.711,422.582,399.161,178.800,23.959,153.534
C01619=1094.717,422.829,399.119,178.802,23.969,153.536
C01620=1094.723,423.075,399.077,178.805,23.979,153.538
C01621=1094.729,423.321,399.036,178.808,23.989,153.540
C01622=1094.735,423.568,398.995,178.810,23.998,153.542
C01623=1094.741,423.815,398.953,178.814,24.009,153.544
C01624=1094.747,424.042,398.916,178.816,24.018,153.546
C01625=1094.753,424.270,398.876,178.819,24.027,153.548
C01626=1094.759,424.498,398.838,178.822,24.037,153.550
C01627=1094.764,424.726,398.800,178.824,24.046,153.552
C01628=1094.770,424.954,398.762,178.827,24.056,153.554
C01629=1094.776,425.182,398.724,178.830,24.065,153.556
C01630=1094.781,425.411,398.685,178.831,24.074,153.558
C01631=1094.787,425.638,398.646,178.834,24.084,153.560
C01632=1094.794,425.884,398.605,178.837,24.094,153.562
C01633=1094.800,426.131,398.563,178.840,24.105,153.565
C01634=1094.806,426.377,398.522,178.843,24.115,153.567
C01635=1094.812,426.624,398.480,178.846,24.125,153.569
C01636=1094.818,426.870,398.439,178.848,24.135,153.571
C01637=1094.825,427.117,398.397,178.852,24.146,153.573
C01638=1094.831,427.363,398.355,178.854,24.156,153.576
C01639=1094.838,427.609,398.313,178.857,24.167,153.578
C01640=1094.844,427.855,398.271,178.860,24.177,153.580
C01641=1094.850,428.102,398.230,178.863,24.188,153.583
C01642=1094.856,428.349,398.188,178.866,24.198,153.585
C01643=1094.862,428.594,398.145,178.868,24.209,153.587
C01644=1094.868,428.841,398.103,178.871,24.220,153.589
C01645=1094.874,429.088,398.062,178.874,24.231,153.592
C01646=1094.881,429.334,398.019,178.877,24.241,153.594
C01647=1094.887,429.580,397.978,178.879,24.252,153.596
C01648=1094.894,429.826,397.935,178.883,24.263,153.599
C01649=1094.899,430.073,397.893,178.885,24.274,153.601
C01650=1094.906,430.319,397.851,178.888,24.285,153.603
C01651=1094.912,430.565,397.809,178.891,24.296,153.606
C01652=1094.919,430.812,397.767,178.894,24.307,153.608
C01653=1094.925,431.058,397.725,178.897,24.318,153.611
C01654=1094.931,431.304,397.682,178.899,24.329,153.613
C01655=1094.937,431.550,397.640,178.902,24.340,153.615
C01656=1094.943,431.797,397.598,178.905,24.351,153.618
C01657=1094.950,432.042,397.556,178.908,24.362,153.620
C01658=1094.956,432.289,397.513,178.911,24.374,153.623
C01659=1094.962,432.535,397.472,178.913,24.385,153.625
C01660=1094.969,432.782,397.429,178.916,24.396,153.628
C01661=1094.974,433.027,397.386,178.919,24.408,153.630
C01662=1094.981,433.274,397.344,178.922,24.419,153.632
C01663=1094.987,433.520,397.301,178.925,24.430,153.635
C01664=1094.993,433.767,397.259,178.927,24.442,153.638
C01665=1095.000,434.013,397.217,178.930,24.454,153.640
C01666=1095.005,434.259,397.174,178.933,24.465,153.643
C01667=1095.012,434.505,397.131,178.936,24.477,153.645
C01668=1095.018,434.751,397.088,178.938,24.488,153.648
C01669=1095.025,434.997,397.046,178.942,24.500,153.650
C01670=1095.031,435.244,397.003,178.944,24.512,153.653
C01671=1095.036,435.490,396.960,178.947,24.524,153.656
C01672=1095.043,435.736,396.917,178.949,24.535,153.658
C01673=1095.049,435.983,396.874,178.952,24.547,153.661
C01674=1095.056,436.228,396.831,178.956,24.559,153.663
C01675=1095.062,436.474,396.788,178.958,24.571,153.666
C01676=1095.069,436.720,396.746,178.961,24.583,153.669
C01677=1095.074,436.966,396.703,178.963,24.595,153.671
C01678=1095.081,437.213,396.660,178.967,24.607,153.674
C01679=1095.088,437.459,396.617,178.970,24.619,153.677
C01680=1095.094,437.699,396.575,178.972,24.631,153.679
C01681=1095.099,437.939,396.533,178.974,24.643,153.682
C01682=1095.106,438.179,396.491,178.978,24.655,153.685
C01683=1095.113,438.420,396.449,178.980,24.667,153.687
C01684=1095.118,438.661,396.407,178.983,24.679,153.690
C01685=1095.125,438.901,396.364,178.985,24.691,153.693
C01686=1095.131,439.141,396.322,178.988,24.703,153.695
C01687=1095.137,439.382,396.280,178.991,24.715,153.698
C01688=1095.144,439.628,396.238,178.994,24.728,153.701
C01689=1095.150,439.874,396.194,178.997,24.740,153.704
C01690=1095.156,440.121,396.151,179.000,24.753,153.706
C01691=1095.163,440.367,396.107,179.002,24.765,153.709
C01692=1095.169,440.612,396.064,179.005,24.778,153.712
C01693=1095.175,440.858,396.021,179.008,24.791,153.715
C01694=1095.182,441.104,395.977,179.010,24.803,153.718
C01695=1095.188,441.350,395.933,179.013,24.816,153.721
C01696=1095.194,441.597,395.890,179.016,24.830,153.724
C01697=1095.201,441.842,395.847,179.019,24.842,153.727
C01698=1095.207,442.088,395.803,179.022,24.855,153.730
C01699=1095.214,442.334,395.759,179.024,24.868,153.732
C01700=1095.220,442.580,395.716,179.027,24.881,153.735
C01701=1095.226,442.826,395.672,179.030,24.895,153.738
C01702=1095.233,443.072,395.628,179.033,24.908,153.741
C01703=1095.239,443.318,395.585,179.036,24.921,153.744
C01704=1095.246,443.564,395.541,179.038,24.934,153.747
C01705=1095.252,443.810,395.497,179.041,24.948,153.750
C01706=1095.259,444.056,395.453,179.044,24.961,153.754
C01707=1095.265,444.302,395.409,179.047,24.975,153.757
C01708=1095.271,444.548,395.365,179.049,24.988,153.760
C01709=1095.278,444.794,395.321,179.051,25.001,153.763
C01710=1095.284,445.040,395.278,179.053,25.014,153.766
C01711=1095.291,445.286,395.234,179.054,25.028,153.769
C01712=1095.297,445.531,395.189,179.056,25.041,153.772
C01713=1095.304,445.777,395.145,179.058,25.054,153.775
C01714=1095.310,446.023,395.102,179.059,25.067,153.779
C01715=1095.317,446.269,395.058,179.060,25.080,153.782
C01716=1095.322,446.516,395.013,179.061,25.094,153.785
C01717=1095.329,446.761,394.969,179.062,25.107,153.788
C01718=1095.336,447.007,394.925,179.063,25.120,153.791
C01719=1095.342,447.253,394.881,179.064,25.133,153.795
C01720=1095.348,447.499,394.837,179.064,25.147,153.798
C01721=1095.354,447.745,394.792,179.064,25.160,153.801
C01722=1095.361,447.991,394.748,179.065,25.173,153.805
C01723=1095.368,448.237,394.704,179.065,25.186,153.808
C01724=1095.375,448.483,394.659,179.065,25.200,153.811
C01725=1095.381,448.729,394.615,179.064,25.212,153.815
C01726=1095.387,448.974,394.570,179.064,25.225,153.818
C01727=1095.393,449.220,394.526,179.064,25.239,153.821
C01728=1095.400,449.466,394.483,179.063,25.251,153.825
C01729=1095.407,449.712,394.438,179.062,25.265,153.828
C01730=1095.413,449.957,394.393,179.061,25.277,153.832
C01731=1095.421,450.203,394.350,179.060,25.290,153.835
C01732=1095.031,450.195,394.181,179.006,25.499,153.895
C01733=1095.022,449.948,394.226,179.006,25.488,153.891
C01734=1095.016,449.702,394.270,179.007,25.474,153.888
C01735=1095.010,449.457,394.315,179.008,25.461,153.885
C01736=1095.003,449.211,394.360,179.009,25.448,153.881
C01737=1094.997,448.965,394.403,179.009,25.435,153.878
C01738=1094.990,448.720,394.448,179.009,25.422,153.874
C01739=1094.983,448.474,394.492,179.010,25.409,153.871
C01740=1094.977,448.228,394.537,179.010,25.396,153.868
C01741=1094.970,447.982,394.581,179.010,25.383,153.864
C01742=1094.964,447.736,394.626,179.010,25.369,153.861
C01743=1094.957,447.490,394.670,179.009,25.356,153.858
C01744=1094.952,447.244,394.714,179.008,25.343,153.854
C01745=1094.945,446.999,394.759,179.008,25.329,153.851
C01746=1094.938,446.753,394.802,179.006,25.316,153.848
C01747=1094.932,446.507,394.846,179.005,25.302,153.845
C01748=1094.925,446.261,394.891,179.004,25.289,153.841
C01749=1094.919,446.014,394.936,179.003,25.276,153.838
C01750=1094.913,445.768,394.979,179.002,25.263,153.835
C01751=1094.906,445.522,395.023,179.000,25.249,153.832
C01752=1094.899,445.277,395.068,178.998,25.236,153.829
C01753=1094.893,445.031,395.112,178.997,25.223,153.825
C01754=1094.887,444.785,395.156,178.994,25.209,153.822
C01755=1094.880,444.539,395.199,178.992,25.196,153.819
C01756=1094.874,444.293,395.243,178.990,25.183,153.816
C01757=1094.867,444.047,395.287,178.987,25.169,153.813
C01758=1094.861,443.801,395.331,178.984,25.156,153.810
C01759=1094.854,443.555,395.375,178.981,25.142,153.807
C01760=1094.848,443.309,395.419,178.979,25.129,153.804
C01761=1094.842,443.063,395.463,178.976,25.116,153.801
C01762=1094.835,442.817,395.506,178.973,25.102,153.798
C01763=1094.829,442.571,395.550,178.970,25.089,153.795
C01764=1094.822,442.325,395.594,178.967,25.076,153.792
C01765=1094.816,442.079,395.638,178.965,25.063,153.789
C01766=1094.810,441.833,395.682,178.962,25.050,153.786
C01767=1094.804,441.588,395.725,178.959,25.037,153.783
C01768=1094.797,441.342,395.769,178.956,25.024,153.780
C01769=1094.790,441.096,395.812,178.953,25.011,153.777
C01770=1094.784,440.850,395.856,178.950,24.998,153.774
C01771=1094.778,440.604,395.899,178.947,24.985,153.772
C01772=1094.771,440.357,395.943,178.944,24.973,153.769
C01773=1094.764,440.112,395.986,178.942,24.960,153.766
C01774=1094.758,439.866,396.030,178.939,24.947,153.763
C01775=1094.752,439.620,396.072,178.936,24.935,153.760
C01776=1094.746,439.374,396.116,178.933,24.922,153.757
C01777=1094.739,439.138,396.158,178.930,24.910,153.755
C01778=1094.733,438.903,396.198,178.928,24.899,153.752
C01779=1094.728,438.668,396.240,178.925,24.887,153.749
C01780=1094.721,438.432,396.281,178.922,24.875,153.747
C01781=1094.714,438.197,396.323,178.919,24.863,153.744
C01782=1094.708,437.962,396.364,178.916,24.851,153.742
C01783=1094.703,437.727,396.405,178.914,24.839,153.739
C01784=1094.697,437.492,396.446,178.911,24.828,153.736
C01785=1094.691,437.245,396.489,178.908,24.815,153.734
C01786=1094.683,436.999,396.532,178.906,24.804,153.731
C01787=1094.677,436.753,396.575,178.902,24.791,153.728
C01788=1094.671,436.507,396.618,178.900,24.779,153.726
C01789=1094.665,436.261,396.661,178.897,24.768,153.723
C01790=1094.658,436.015,396.704,178.894,24.755,153.720
C01791=1094.652,435.769,396.747,178.891,24.743,153.718
C01792=1094.646,435.523,396.790,178.888,24.732,153.715
C01793=1094.639,435.276,396.832,178.886,24.720,153.712
C01794=1094.634,435.030,396.875,178.882,24.708,153.710
C01795=1094.627,434.784,396.918,178.880,24.696,153.707
C01796=1094.621,434.537,396.961,178.877,24.684,153.705
C01797=1094.615,434.292,397.003,178.874,24.673,153.702
C01798=1094.608,434.045,397.046,178.871,24.661,153.700
C01799=1094.602,433.800,397.088,178.868,24.649,153.697
C01800=1094.596,433.553,397.132,178.865,24.638,153.694
C01801=1094.589,433.307,397.174,178.863,24.627,153.692
C01802=1094.584,433.061,397.217,178.859,24.615,153.689
C01803=1094.577,432.815,397.259,178.857,24.604,153.687
C01804=1094.571,432.569,397.302,178.854,24.592,153.685
C01805=1094.565,432.322,397.344,178.851,24.581,153.682
C01806=1094.558,432.076,397.386,178.848,24.570,153.680
C01807=1094.552,431.830,397.429,178.845,24.558,153.677
C01808=1094.545,431.584,397.471,178.843,24.547,153.675
C01809=1094.540,431.337,397.513,178.839,24.536,153.672
C01810=1094.533,431.091,397.556,178.837,24.525,153.670
C01811=1094.526,430.845,397.598,178.834,24.514,153.668
C01812=1094.520,430.598,397.640,178.831,24.503,153.665
C01813=1094.514,430.353,397.683,178.828,24.492,153.663
C01814=1094.508,430.106,397.724,178.825,24.481,153.660
C01815=1094.502,429.860,397.767,178.822,24.469,153.658
